C01843=1138.601,45.378,-51.505,-179.902,6.447,149.146
C01844=1138.595,45.628,-51.520,-179.900,6.448,149.145
C01845=1138.590,45.878,-51.536,-179.897,6.449,149.145
C01846=1138.585,46.127,-51.551,-179.895,6.450,149.144
C01847=1138.580,46.377,-51.567,-179.892,6.451,149.144
C01848=1138.576,46.626,-51.582,-179.890,6.452,149.143
C01849=1138.570,46.875,-51.597,-179.886,6.453,149.143
C01850=1138.565,47.125,-51.613,-179.884,6.454,149.142
C01851=1138.560,47.374,-51.628,-179.881,6.456,149.142
C01852=1138.556,47.624,-51.644,-179.879,6.456,149.141
C01853=1138.550,47.873,-51.659,-179.876,6.458,149.141
C01854=1138.546,48.122,-51.674,-179.873,6.460,149.140
C01855=1138.540,48.372,-51.690,-179.871,6.460,149.140
C01856=1138.535,48.621,-51.706,-179.868,6.462,149.139
C01857=1138.531,48.871,-51.721,-179.866,6.463,149.139
C01858=1138.525,49.120,-51.736,-179.863,6.464,149.138
C01859=1138.520,49.370,-51.752,-179.860,6.465,149.138
C01860=1138.515,49.619,-51.767,-179.858,6.466,149.137
C01861=1138.510,49.869,-51.783,-179.855,6.467,149.137
C01862=1138.505,50.118,-51.799,-179.852,6.468,149.136
C01863=1138.500,50.368,-51.814,-179.850,6.469,149.136
C01864=1138.495,50.617,-51.829,-179.847,6.471,149.135
C01865=1138.490,50.867,-51.845,-179.844,6.472,149.135
C01866=1138.485,51.116,-51.861,-179.842,6.473,149.134
C01867=1138.480,51.365,-51.876,-179.839,6.474,149.133
C01868=1138.475,51.616,-51.892,-179.837,6.475,149.133
C01869=1138.470,51.865,-51.907,-179.834,6.477,149.133
C01870=1138.465,52.114,-51.923,-179.831,6.477,149.132
C01871=1138.459,52.364,-51.938,-179.828,6.479,149.131
C01872=1138.456,52.613,-51.954,-179.826,6.480,149.131
C01873=1138.450,52.862,-51.970,-179.823,6.481,149.131
C01874=1138.445,53.131,-51.987,-179.820,6.483,149.130
C01875=1138.439,53.399,-52.004,-179.817,6.484,149.129
C01876=1138.433,53.668,-52.020,-179.815,6.485,149.129
C01877=1138.428,53.938,-52.038,-179.812,6.486,149.128
C01878=1138.423,54.186,-52.054,-179.809,6.488,149.128
C01879=1138.418,54.435,-52.069,-179.807,6.488,149.127
C01880=1138.414,54.686,-52.085,-179.804,6.490,149.127
C01881=1138.408,54.935,-52.101,-179.801,6.491,149.126
C01882=1138.403,55.184,-52.116,-179.799,6.492,149.126
C01883=1138.398,55.434,-52.133,-179.796,6.494,149.125
C01884=1138.393,55.683,-52.148,-179.793,6.494,149.125
C01885=1138.388,55.933,-52.164,-179.790,6.496,149.124
C01886=1138.384,56.182,-52.179,-179.788,6.497,149.124
C01887=1138.379,56.431,-52.196,-179.785,6.498,149.123
C01888=1138.373,56.681,-52.211,-179.782,6.500,149.123
C01889=1138.368,56.931,-52.227,-179.780,6.501,149.122
C01890=1138.363,57.180,-52.244,-179.777,6.502,149.122
C01891=1138.359,57.430,-52.260,-179.775,6.503,149.121
C01892=1138.353,57.679,-52.275,-179.772,6.504,149.121
C01893=1138.348,57.928,-52.291,-179.769,6.506,149.120
C01894=1138.343,58.178,-52.307,-179.767,6.506,149.119
C01895=1138.338,58.427,-52.323,-179.764,6.508,149.119
C01896=1138.333,58.676,-52.339,-179.762,6.509,149.119
C01897=1138.328,58.926,-52.355,-179.759,6.511,149.118
C01898=1138.323,59.175,-52.372,-179.756,6.512,149.117
C01899=1138.318,59.425,-52.387,-179.753,6.513,149.117
C01900=1138.313,59.675,-52.403,-179.751,6.514,149.117
C01901=1138.308,59.924,-52.420,-179.747,6.516,149.116
C01902=1138.303,60.173,-52.435,-179.745,6.516,149.116
C01903=1138.298,60.422,-52.452,-179.743,6.518,149.115
C01904=1138.293,60.672,-52.468,-179.740,6.519,149.115
C01905=1138.288,60.921,-52.484,-179.737,6.520,149.114
C01906=1138.283,61.171,-52.500,-179.734,6.522,149.114
C01907=1138.278,61.420,-52.516,-179.732,6.523,149.113
C01908=1138.273,61.670,-52.532,-179.729,6.524,149.112
C01909=1138.268,61.919,-52.548,-179.726,6.526,149.112
C01910=1138.263,62.169,-52.564,-179.724,6.526,149.112
C01911=1138.258,62.418,-52.581,-179.721,6.528,149.111
C01912=1138.254,62.668,-52.597,-179.719,6.529,149.110
C01913=1138.248,62.917,-52.613,-179.716,6.530,149.110
C01914=1138.244,63.167,-52.629,-179.713,6.532,149.110
C01915=1138.239,63.416,-52.645,-179.711,6.532,149.109
C01916=1138.234,63.666,-52.661,-179.708,6.534,149.108
C01917=1138.229,63.914,-52.677,-179.705,6.536,149.108
C01918=1138.224,64.164,-52.694,-179.703,6.536,149.108
C01919=1138.219,64.413,-52.710,-179.700,6.538,149.107
C01920=1138.214,64.663,-52.727,-179.697,6.539,149.106
C01921=1138.208,64.912,-52.743,-179.695,6.540,149.106
C01922=1138.204,65.162,-52.759,-179.692,6.542,149.105
C01923=1138.199,65.411,-52.776,-179.689,6.543,149.105
C01924=1138.194,65.661,-52.791,-179.687,6.544,149.105
C01925=1138.189,65.910,-52.808,-179.684,6.546,149.104
C01926=1138.184,66.159,-52.824,-179.681,6.547,149.103
C01927=1138.178,66.409,-52.841,-179.679,6.548,149.103
C01928=1138.174,66.658,-52.857,-179.676,6.549,149.103
C01929=1138.169,66.908,-52.874,-179.673,6.551,149.102
C01930=1138.164,67.157,-52.890,-179.670,6.552,149.101
C01931=1138.159,67.407,-52.906,-179.668,6.553,149.101
C01932=1138.154,67.655,-52.923,-179.665,6.555,149.101
C01933=1138.149,67.905,-52.940,-179.662,6.555,149.100
C01934=1138.144,68.154,-52.956,-179.659,6.557,149.099
C01935=1138.139,68.404,-52.972,-179.657,6.559,149.099
C01936=1138.135,68.654,-52.989,-179.655,6.559,149.099
C01937=1138.129,68.903,-53.006,-179.651,6.561,149.098
C01938=1138.124,69.152,-53.022,-179.649,6.562,149.098
C01939=1138.119,69.402,-53.038,-179.646,6.564,149.097
C01940=1138.115,69.651,-53.055,-179.644,6.565,149.097
C01941=1138.109,69.901,-53.072,-179.640,6.566,149.096
C01942=1138.104,70.150,-53.088,-179.638,6.568,149.096
C01943=1138.100,70.399,-53.105,-179.636,6.569,149.095
C01944=1138.095,70.648,-53.121,-179.633,6.570,149.095
C01945=1138.089,70.898,-53.138,-179.630,6.572,149.094
C01946=1138.085,71.148,-53.154,-179.627,6.572,149.094
C01947=1138.080,71.397,-53.171,-179.625,6.574,149.093
C01948=1138.074,71.646,-53.188,-179.622,6.576,149.093
C01949=1138.070,71.896,-53.205,-179.619,6.577,149.092
C01950=1138.065,72.145,-53.221,-179.617,6.578,149.092
C01951=1138.060,72.394,-53.238,-179.614,6.580,149.091
C01952=1138.055,72.644,-53.255,-179.611,6.581,149.091
C01953=1138.050,72.893,-53.271,-179.608,6.582,149.090
C01954=1138.045,73.143,-53.288,-179.606,6.583,149.090
C01955=1138.040,73.392,-53.305,-179.603,6.585,149.089
C01956=1138.035,73.641,-53.321,-179.600,6.587,149.089
C01957=1138.030,73.891,-53.339,-179.598,6.587,149.088
C01958=1138.026,74.140,-53.355,-179.595,6.589,149.088
C01959=1138.020,74.389,-53.372,-179.592,6.590,149.087
C01960=1138.015,74.639,-53.389,-179.590,6.591,149.087
C01961=1138.011,74.888,-53.405,-179.587,6.593,149.086
C01962=1138.006,75.138,-53.423,-179.584,6.594,149.086
C01963=1138.001,75.387,-53.439,-179.581,6.596,149.085
C01964=1137.995,75.637,-53.456,-179.579,6.597,149.085
C01965=1137.991,75.886,-53.473,-179.576,6.598,149.084
C01966=1137.985,76.135,-53.490,-179.573,6.600,149.084
C01967=1137.981,76.385,-53.507,-179.570,6.601,149.083
C01968=1137.976,76.634,-53.523,-179.568,6.602,149.083
C01969=1137.971,76.884,-53.540,-179.565,6.604,149.082
C01970=1137.966,77.132,-53.557,-179.562,6.605,149.082
C01971=1137.961,77.382,-53.575,-179.559,6.607,149.081
C01972=1137.956,77.631,-53.591,-179.557,6.608,149.081
C01973=1137.951,77.881,-53.609,-179.555,6.609,149.081
C01974=1137.946,78.130,-53.625,-179.551,6.611,149.080
C01975=1137.941,78.380,-53.642,-179.549,6.612,149.080
C01976=1137.937,78.629,-53.660,-179.546,6.613,149.079
C01977=1137.931,78.878,-53.677,-179.544,6.615,149.079
C01978=1137.926,79.146,-53.695,-179.540,6.616,149.078
C01979=1137.921,79.415,-53.713,-179.538,6.618,149.078
C01980=1137.915,79.684,-53.732,-179.535,6.619,149.077
C01981=1137.910,79.952,-53.750,-179.532,6.621,149.077
C01982=1137.905,80.202,-53.767,-179.529,6.622,149.076
C01983=1137.901,80.450,-53.784,-179.526,6.624,149.076
C01984=1137.896,80.700,-53.802,-179.524,6.624,149.075
C01985=1137.890,80.949,-53.819,-179.521,6.626,149.075
C01986=1137.885,81.199,-53.835,-179.518,6.628,149.074
C01987=1137.880,81.448,-53.853,-179.515,6.629,149.074
C01988=1137.876,81.698,-53.870,-179.513,6.631,149.073
C01989=1137.871,81.947,-53.887,-179.510,6.632,149.073
C01990=1137.866,82.196,-53.905,-179.507,6.633,149.072
C01991=1137.861,82.445,-53.921,-179.505,6.635,149.072
C01992=1137.855,82.695,-53.939,-179.502,6.637,149.071
C01993=1137.851,82.944,-53.957,-179.499,6.637,149.071
C01994=1137.846,83.194,-53.973,-179.496,6.639,149.070
C01995=1137.841,83.443,-53.991,-179.494,6.640,149.070
C01996=1137.837,83.692,-54.008,-179.491,6.642,149.069
C01997=1137.831,83.942,-54.025,-179.488,6.644,149.069
C01998=1137.826,84.191,-54.043,-179.486,6.644,149.068
C01999=1137.821,84.440,-54.060,-179.483,6.646,149.068
C02000=1137.817,84.689,-54.078,-179.480,6.648,149.068
C02001=1137.811,84.939,-54.095,-179.477,6.649,149.067
C02002=1137.806,85.188,-54.113,-179.475,6.651,149.067
C02003=1137.802,85.438,-54.129,-179.472,6.651,149.066
C02004=1137.797,85.687,-54.147,-179.469,6.653,149.066
C02005=1137.792,85.937,-54.165,-179.466,6.655,149.065
C02006=1137.788,86.186,-54.182,-179.464,6.656,149.065
C02007=1137.782,86.435,-54.199,-179.461,6.658,149.064
C02008=1137.778,86.685,-54.217,-179.458,6.659,149.064
C02009=1137.772,86.934,-54.234,-179.456,6.660,149.063
C02010=1137.768,87.183,-54.252,-179.453,6.662,149.063
C02011=1137.762,87.432,-54.269,-179.450,6.663,149.062
C02012=1137.757,87.681,-54.287,-179.447,6.665,149.062
C02013=1137.752,87.931,-54.304,-179.444,6.666,149.061
C02014=1137.747,88.180,-54.322,-179.441,6.668,149.061
C02015=1137.743,88.429,-54.339,-179.439,6.669,149.060
C02016=1137.738,88.679,-54.357,-179.437,6.671,149.060
C02017=1137.733,88.928,-54.375,-179.434,6.672,149.060
C02018=1137.728,89.178,-54.392,-179.431,6.674,149.059
C02019=1137.723,89.427,-54.410,-179.428,6.675,149.059
C02020=1137.719,89.676,-54.427,-179.425,6.677,149.058
C02021=1137.713,89.926,-54.445,-179.423,6.678,149.058
C02022=1137.709,90.175,-54.463,-179.420,6.679,149.057
C02023=1137.704,90.424,-54.481,-179.417,6.681,149.057
C02024=1137.698,90.674,-54.498,-179.414,6.682,149.056
C02025=1137.693,90.923,-54.516,-179.412,6.684,149.056
C02026=1137.689,91.172,-54.534,-179.409,6.686,149.055
C02027=1137.684,91.421,-54.551,-179.406,6.687,149.055
C02028=1137.679,91.671,-54.568,-179.404,6.688,149.055
C02029=1137.674,91.920,-54.586,-179.401,6.690,149.054
C02030=1137.669,92.169,-54.604,-179.398,6.691,149.053
C02031=1137.664,92.419,-54.622,-179.395,6.693,149.053
C02032=1137.659,92.668,-54.640,-179.392,6.695,149.053
C02033=1137.654,92.918,-54.658,-179.390,6.696,149.052
C02034=1137.649,93.167,-54.676,-179.387,6.698,149.052
C02035=1137.644,93.416,-54.694,-179.385,6.699,149.051
C02036=1137.640,93.665,-54.712,-179.382,6.700,149.051
C02037=1137.635,93.916,-54.729,-179.379,6.702,149.050
C02038=1137.630,94.165,-54.747,-179.376,6.703,149.050
C02039=1137.625,94.414,-54.765,-179.373,6.705,149.049
C02040=1137.620,94.663,-54.783,-179.371,6.707,149.049
C02041=1137.615,94.912,-54.801,-179.368,6.708,149.049
C02042=1137.610,95.161,-54.819,-179.365,6.710,149.048
C02043=1137.605,95.411,-54.837,-179.362,6.711,149.048
C02044=1137.600,95.660,-54.854,-179.360,6.712,149.047
C02045=1137.595,95.910,-54.872,-179.357,6.714,149.047
C02046=1137.590,96.159,-54.890,-179.354,6.716,149.046
C02047=1137.586,96.408,-54.908,-179.352,6.717,149.046
C02048=1137.581,96.658,-54.927,-179.349,6.719,149.045
C02049=1137.576,96.907,-54.945,-179.346,6.720,149.045
C02050=1137.571,97.156,-54.963,-179.343,6.722,149.044
C02051=1137.566,97.405,-54.981,-179.340,6.724,149.044
C02052=1137.562,97.655,-54.999,-179.337,6.725,149.044
C02053=1137.557,97.904,-55.017,-179.335,6.726,149.043
C02054=1137.552,98.153,-55.035,-179.333,6.728,149.043
C02055=1137.547,98.403,-55.053,-179.330,6.729,149.042
C02056=1137.543,98.652,-55.071,-179.327,6.731,149.042
C02057=1137.538,98.901,-55.089,-179.324,6.732,149.041
C02058=1137.532,99.151,-55.107,-179.321,6.734,149.041
C02059=1137.527,99.400,-55.125,-179.318,6.736,149.040
C02060=1137.522,99.649,-55.143,-179.316,6.737,149.040
C02061=1137.518,99.898,-55.162,-179.313,6.739,149.040
C02062=1137.513,100.147,-55.180,-179.310,6.741,149.039
C02063=1137.508,100.397,-55.198,-179.307,6.742,149.039
C02064=1137.503,100.646,-55.216,-179.304,6.744,149.038
C02065=1137.498,100.895,-55.235,-179.301,6.745,149.038
C02066=1137.493,101.145,-55.253,-179.299,6.746,149.037
C02067=1137.489,101.394,-55.271,-179.297,6.748,149.037
C02068=1137.484,101.643,-55.289,-179.294,6.750,149.036
C02069=1137.479,101.892,-55.308,-179.291,6.751,149.036
C02070=1137.474,102.141,-55.326,-179.288,6.753,149.036
C02071=1137.469,102.391,-55.345,-179.286,6.755,149.035
C02072=1137.464,102.641,-55.363,-179.282,6.756,149.035
C02073=1137.459,102.890,-55.381,-179.280,6.758,149.034
C02074=1137.455,103.138,-55.399,-179.277,6.759,149.034
C02075=1137.450,103.389,-55.418,-179.274,6.761,149.033
C02076=1137.445,103.638,-55.436,-179.272,6.763,149.033
C02077=1137.440,103.887,-55.454,-179.269,6.764,149.033
C02078=1137.435,104.135,-55.473,-179.266,6.766,149.032
C02079=1137.430,104.386,-55.492,-179.263,6.768,149.032
C02080=1137.425,104.635,-55.510,-179.261,6.769,149.031
C02081=1137.421,104.883,-55.529,-179.257,6.771,149.031
C02082=1137.415,105.152,-55.549,-179.255,6.772,149.030
C02083=1137.410,105.421,-55.568,-179.252,6.774,149.030
C02084=1137.404,105.689,-55.588,-179.249,6.776,149.029
C02085=1137.400,105.957,-55.609,-179.246,6.777,149.029
C02086=1137.395,106.206,-55.627,-179.243,6.779,149.028
C02087=1137.390,106.456,-55.646,-179.240,6.780,149.028
C02088=1137.385,106.705,-55.664,-179.238,6.782,149.028
C02089=1137.380,106.954,-55.682,-179.235,6.784,149.027
C02090=1137.375,107.204,-55.702,-179.232,6.785,149.027
C02091=1137.371,107.453,-55.720,-179.230,6.787,149.026
C02092=1137.366,107.702,-55.738,-179.227,6.789,149.026
C02093=1137.361,107.952,-55.757,-179.224,6.790,149.025
C02094=1137.356,108.201,-55.775,-179.221,6.792,149.025
C02095=1137.351,108.450,-55.795,-179.218,6.793,149.024
C02096=1137.346,108.700,-55.813,-179.215,6.795,149.024
C02097=1137.342,108.948,-55.832,-179.213,6.797,149.024
C02098=1137.336,109.198,-55.850,-179.210,6.798,149.023
C02099=1137.332,109.447,-55.869,-179.207,6.800,149.023
C02100=1137.326,109.696,-55.888,-179.204,6.802,149.022
C02101=1137.322,109.946,-55.907,-179.202,6.804,149.022
C02102=1137.317,110.195,-55.926,-179.199,6.805,149.022
C02103=1137.312,110.444,-55.944,-179.196,6.807,149.021
C02104=1137.308,110.694,-55.963,-179.194,6.809,149.021
C02105=1137.302,110.942,-55.982,-179.191,6.810,149.020
C02106=1137.298,111.192,-56.001,-179.188,6.812,149.020
C02107=1137.293,111.441,-56.020,-179.185,6.813,149.019
C02108=1137.288,111.690,-56.038,-179.182,6.815,149.019
C02109=1137.283,111.940,-56.057,-179.179,6.817,149.019
C02110=1137.279,112.188,-56.076,-179.177,6.818,149.018
C02111=1137.274,112.438,-56.096,-179.174,6.820,149.018
C02112=1137.269,112.687,-56.114,-179.171,6.822,149.017
C02113=1137.264,112.936,-56.133,-179.168,6.823,149.017
C02114=1137.259,113.186,-56.153,-179.166,6.825,149.016
C02115=1137.254,113.435,-56.171,-179.163,6.827,149.016
C02116=1137.249,113.684,-56.190,-179.160,6.828,149.016
C02117=1137.245,113.933,-56.209,-179.158,6.830,149.015
C02118=1137.240,114.183,-56.228,-179.154,6.833,149.015
C02119=1137.235,114.432,-56.246,-179.152,6.834,149.014
C02120=1137.230,114.681,-56.266,-179.149,6.836,149.014
C02121=1137.225,114.930,-56.285,-179.146,6.838,149.014
C02122=1137.221,115.180,-56.304,-179.143,6.839,149.013
C02123=1137.215,115.429,-56.323,-179.141,6.841,149.013
C02124=1137.211,115.678,-56.342,-179.137,6.842,149.012
C02125=1137.206,115.927,-56.361,-179.135,6.844,149.012
C02126=1137.201,116.177,-56.381,-179.132,6.846,149.011
C02127=1137.196,116.426,-56.399,-179.129,6.847,149.011
C02128=1137.191,116.675,-56.419,-179.126,6.849,149.011
C02129=1137.186,116.924,-56.438,-179.124,6.851,149.010
C02130=1137.182,117.173,-56.457,-179.121,6.852,149.010
C02131=1137.177,117.422,-56.476,-179.118,6.854,149.009
C02132=1137.172,117.672,-56.496,-179.116,6.856,149.009
C02133=1137.167,117.920,-56.515,-179.113,6.857,149.009
C02134=1137.163,118.170,-56.534,-179.110,6.859,149.008
C02135=1137.157,118.419,-56.553,-179.107,6.861,149.008
C02136=1137.153,118.669,-56.572,-179.105,6.862,149.007
C02137=1137.148,118.918,-56.591,-179.101,6.865,149.007
C02138=1137.143,119.167,-56.611,-179.099,6.867,149.007
C02139=1137.139,119.416,-56.630,-179.096,6.868,149.006
C02140=1137.134,119.665,-56.649,-179.093,6.870,149.006
C02141=1137.129,119.915,-56.669,-179.090,6.872,149.005
C02142=1137.123,120.164,-56.688,-179.088,6.873,149.005
C02143=1137.119,120.413,-56.707,-179.085,6.875,149.005
C02144=1137.114,120.662,-56.727,-179.082,6.877,149.004
C02145=1137.109,120.911,-56.746,-179.079,6.878,149.004
C02146=1137.105,121.161,-56.766,-179.077,6.880,149.003
C02147=1137.099,121.410,-56.785,-179.074,6.882,149.003
C02148=1137.095,121.659,-56.804,-179.071,6.883,149.002
C02149=1137.090,121.908,-56.824,-179.068,6.886,149.002
C02150=1137.085,122.158,-56.843,-179.065,6.888,149.002
C02151=1137.081,122.406,-56.864,-179.063,6.889,149.001
C02152=1137.075,122.655,-56.883,-179.060,6.891,149.001
C02153=1137.071,122.905,-56.902,-179.057,6.893,149.000
C02154=1137.067,123.154,-56.922,-179.054,6.894,149.000
C02155=1137.061,123.403,-56.941,-179.052,6.896,149.000
C02156=1137.057,123.653,-56.961,-179.049,6.898,148.999
C02157=1137.052,123.902,-56.980,-179.046,6.899,148.999
C02158=1137.046,124.151,-56.999,-179.043,6.901,148.998
C02159=1137.042,124.400,-57.020,-179.040,6.904,148.998
C02160=1137.038,124.649,-57.039,-179.037,6.905,148.998
C02161=1137.033,124.898,-57.058,-179.035,6.907,148.997
C02162=1137.028,125.148,-57.078,-179.032,6.909,148.997
C02163=1137.024,125.397,-57.098,-179.029,6.910,148.996
C02164=1137.018,125.645,-57.118,-179.027,6.912,148.996
C02165=1137.013,125.895,-57.137,-179.024,6.914,148.996
C02166=1137.009,126.145,-57.157,-179.021,6.915,148.995
C02167=1137.004,126.394,-57.177,-179.018,6.918,148.995
C02168=1136.999,126.642,-57.197,-179.015,6.920,148.995
C02169=1136.994,126.892,-57.216,-179.012,6.921,148.994
C02170=1136.989,127.142,-57.236,-179.010,6.923,148.994
C02171=1136.984,127.390,-57.256,-179.007,6.925,148.993
C02172=1136.980,127.639,-57.275,-179.004,6.926,148.993
C02173=1136.975,127.889,-57.295,-179.001,6.928,148.993
C02174=1136.970,128.138,-57.316,-178.998,6.931,148.992
C02175=1136.965,128.387,-57.335,-178.995,6.932,148.992
C02176=1136.961,128.636,-57.355,-178.993,6.934,148.991
C02177=1136.956,128.885,-57.375,-178.990,6.936,148.991
C02178=1136.951,129.135,-57.394,-178.987,6.937,148.991
C02179=1136.946,129.383,-57.414,-178.984,6.939,148.990
C02180=1136.941,129.633,-57.434,-178.982,6.941,148.990
C02181=1136.937,129.882,-57.455,-178.978,6.943,148.989
C02182=1136.932,130.131,-57.474,-178.976,6.945,148.989
C02183=1136.927,130.380,-57.493,-178.973,6.947,148.989
C02184=1136.922,130.629,-57.514,-178.970,6.948,148.988
C02185=1136.918,130.879,-57.533,-178.968,6.950,148.988
C02186=1136.912,131.147,-57.556,-178.964,6.953,148.987
C02187=1136.907,131.416,-57.577,-178.961,6.954,148.987
C02188=1136.903,131.684,-57.598,-178.959,6.956,148.987
C02189=1136.897,131.953,-57.620,-178.955,6.958,148.986
C02190=1136.892,132.202,-57.640,-178.953,6.960,148.986
C02191=1136.888,132.451,-57.660,-178.950,6.962,148.985
C02192=1136.883,132.700,-57.680,-178.947,6.964,148.985
C02193=1136.878,132.949,-57.700,-178.944,6.966,148.985
C02194=1136.873,133.198,-57.721,-178.941,6.968,148.984
C02195=1136.868,133.448,-57.741,-178.939,6.969,148.984
C02196=1136.864,133.697,-57.761,-178.936,6.971,148.983
C02197=1136.859,133.946,-57.781,-178.934,6.973,148.983
C02198=1136.855,134.195,-57.801,-178.930,6.976,148.983
C02199=1136.850,134.443,-57.821,-178.928,6.977,148.983
C02200=1136.844,134.693,-57.841,-178.925,6.979,148.982
C02201=1136.840,134.942,-57.862,-178.922,6.981,148.982
C02202=1136.835,135.191,-57.882,-178.919,6.982,148.981
C02203=1136.831,135.441,-57.902,-178.916,6.985,148.981
C02204=1136.825,135.690,-57.923,-178.913,6.987,148.981
C02205=1136.821,135.939,-57.943,-178.911,6.988,148.980
C02206=1136.816,136.189,-57.963,-178.908,6.990,148.980
C02207=1136.812,136.438,-57.983,-178.905,6.992,148.979
C02208=1136.806,136.686,-58.004,-178.902,6.994,148.979
C02209=1136.802,136.935,-58.024,-178.899,6.996,148.979
C02210=1136.797,137.185,-58.044,-178.897,6.998,148.978
C02211=1136.792,137.434,-58.064,-178.894,7.000,148.978
C02212=1136.787,137.683,-58.085,-178.891,7.001,148.978
C02213=1136.783,137.932,-58.106,-178.888,7.004,148.977
C02214=1136.778,138.181,-58.126,-178.885,7.006,148.977
C02215=1136.773,138.431,-58.146,-178.883,7.007,148.976
C02216=1136.768,138.680,-58.167,-178.880,7.009,148.976
C02217=1136.764,138.928,-58.187,-178.877,7.011,148.976
C02218=1136.759,139.178,-58.208,-178.874,7.013,148.975
C02219=1136.754,139.427,-58.228,-178.871,7.015,148.975
C02220=1136.750,139.676,-58.249,-178.869,7.017,148.975
C02221=1136.745,139.925,-58.270,-178.866,7.019,148.974
C02222=1136.740,140.174,-58.290,-178.863,7.021,148.974
C02223=1136.736,140.423,-58.310,-178.860,7.023,148.974
C02224=1136.730,140.673,-58.331,-178.857,7.025,148.973
C02225=1136.726,140.922,-58.351,-178.855,7.026,148.973
C02226=1136.721,141.171,-58.372,-178.851,7.029,148.972
C02227=1136.716,141.420,-58.392,-178.849,7.030,148.972
C02228=1136.712,141.669,-58.413,-178.846,7.032,148.972
C02229=1136.707,141.918,-58.434,-178.844,7.034,148.971
C02230=1136.702,142.167,-58.454,-178.840,7.037,148.971
C02231=1136.697,142.416,-58.475,-178.838,7.038,148.971
C02232=1136.693,142.665,-58.495,-178.835,7.040,148.970
C02233=1136.687,142.914,-58.516,-178.832,7.043,148.970
C02234=1136.683,143.163,-58.537,-178.829,7.044,148.970
C02235=1136.678,143.412,-58.558,-178.826,7.046,148.969
C02236=1136.674,143.661,-58.579,-178.824,7.048,148.969
C02237=1136.669,143.910,-58.599,-178.821,7.051,148.969
C02238=1136.664,144.159,-58.620,-178.818,7.052,148.968
C02239=1136.660,144.408,-58.640,-178.815,7.054,148.968
C02240=1136.655,144.658,-58.662,-178.813,7.056,148.967
C02241=1136.650,144.907,-58.683,-178.809,7.058,148.967
C02242=1136.646,145.156,-58.703,-178.807,7.060,148.967
C02243=1136.640,145.406,-58.724,-178.804,7.062,148.967
C02244=1136.636,145.654,-58.745,-178.801,7.064,148.966
C02245=1136.631,145.903,-58.766,-178.798,7.066,148.966
C02246=1136.627,146.152,-58.787,-178.796,7.068,148.965
C02247=1136.621,146.401,-58.807,-178.793,7.070,148.965
C02248=1136.617,146.650,-58.828,-178.790,7.072,148.965
C02249=1136.612,146.899,-58.850,-178.787,7.074,148.964
C02250=1136.608,147.149,-58.871,-178.785,7.076,148.964
C02251=1136.603,147.398,-58.891,-178.781,7.078,148.964
C02252=1136.598,147.647,-58.912,-178.779,7.080,148.963
C02253=1136.594,147.895,-58.933,-178.776,7.082,148.963
C02254=1136.589,148.145,-58.954,-178.773,7.083,148.963
C02255=1136.583,148.394,-58.975,-178.770,7.086,148.962
C02256=1136.580,148.643,-58.997,-178.768,7.088,148.962
C02257=1136.575,148.892,-59.018,-178.765,7.090,148.962
C02258=1136.570,149.142,-59.039,-178.762,7.092,148.961
C02259=1136.565,149.390,-59.060,-178.759,7.094,148.961
C02260=1136.560,149.639,-59.081,-178.756,7.096,148.961
C02261=1136.555,149.888,-59.102,-178.753,7.099,148.960
C02262=1136.552,150.137,-59.123,-178.751,7.100,148.960
C02263=1136.546,150.387,-59.144,-178.748,7.102,148.960
C02264=1136.542,150.635,-59.166,-178.745,7.104,148.959
C02265=1136.536,150.885,-59.187,-178.742,7.106,148.959
C02266=1136.532,151.133,-59.207,-178.739,7.108,148.958
C02267=1136.528,151.383,-59.229,-178.736,7.111,148.958
C02268=1136.522,151.632,-59.250,-178.734,7.112,148.958
C02269=1136.518,151.881,-59.272,-178.731,7.114,148.958
C02270=1136.513,152.130,-59.292,-178.728,7.117,148.957
C02271=1136.508,152.378,-59.314,-178.725,7.118,148.957
C02272=1136.504,152.628,-59.335,-178.723,7.120,148.957
C02273=1136.499,152.877,-59.357,-178.719,7.123,148.956
C02274=1136.494,153.126,-59.378,-178.717,7.125,148.956
C02275=1136.490,153.375,-59.399,-178.714,7.126,148.955
C02276=1136.485,153.624,-59.420,-178.711,7.129,148.955
C02277=1136.480,153.873,-59.442,-178.708,7.131,148.955
C02278=1136.475,154.122,-59.463,-178.706,7.133,148.955
C02279=1136.471,154.372,-59.485,-178.702,7.135,148.954
C02280=1136.467,154.620,-59.506,-178.700,7.137,148.954
C02281=1136.461,154.869,-59.527,-178.697,7.139,148.954
C02282=1136.456,155.118,-59.549,-178.694,7.141,148.953
C02283=1136.452,155.367,-59.571,-178.691,7.143,148.953
C02284=1136.447,155.617,-59.592,-178.688,7.146,148.953
C02285=1136.442,155.865,-59.613,-178.685,7.147,148.952
C02286=1136.438,156.115,-59.635,-178.683,7.149,148.952
C02287=1136.433,156.364,-59.656,-178.680,7.152,148.952
C02288=1136.429,156.612,-59.677,-178.677,7.154,148.951
C02289=1136.424,156.861,-59.700,-178.674,7.155,148.951
C02290=1136.419,157.131,-59.723,-178.671,7.158,148.951
C02291=1136.414,157.400,-59.746,-178.668,7.161,148.950
C02292=1136.408,157.668,-59.769,-178.666,7.163,148.950
C02293=1136.403,157.937,-59.793,-178.662,7.165,148.950
C02294=1136.399,158.186,-59.814,-178.660,7.167,148.949
C02295=1136.394,158.436,-59.835,-178.656,7.169,148.949
C02296=1136.390,158.685,-59.857,-178.654,7.171,148.949
C02297=1136.385,158.934,-59.879,-178.651,7.173,148.948
C02298=1136.380,159.182,-59.901,-178.648,7.176,148.948
C02299=1136.376,159.432,-59.923,-178.645,7.177,148.948
C02300=1136.371,159.680,-59.944,-178.642,7.180,148.947
C02301=1136.366,159.929,-59.965,-178.640,7.182,148.947
C02302=1136.362,160.179,-59.987,-178.637,7.184,148.947
C02303=1136.357,160.427,-60.009,-178.634,7.186,148.946
C02304=1136.352,160.677,-60.031,-178.631,7.188,148.946
C02305=1136.348,160.925,-60.053,-178.628,7.191,148.946
C02306=1136.343,161.175,-60.075,-178.625,7.192,148.945
C02307=1136.338,161.424,-60.097,-178.622,7.195,148.945
C02308=1136.333,161.672,-60.119,-178.620,7.197,148.945
C02309=1136.329,161.922,-60.141,-178.617,7.199,148.945
C02310=1136.324,162.170,-60.162,-178.614,7.201,148.944
C02311=1136.319,162.420,-60.184,-178.612,7.203,148.944
C02312=1136.315,162.668,-60.206,-178.608,7.206,148.944
C02313=1136.310,162.918,-60.228,-178.606,7.207,148.943
C02314=1136.305,163.166,-60.250,-178.603,7.209,148.943
C02315=1136.301,163.416,-60.272,-178.600,7.212,148.943
C02316=1136.296,163.664,-60.294,-178.597,7.214,148.942
C02317=1136.291,163.914,-60.316,-178.594,7.216,148.942
C02318=1136.286,164.163,-60.338,-178.592,7.218,148.942
C02319=1136.282,164.412,-60.360,-178.589,7.221,148.942
C02320=1136.277,164.661,-60.382,-178.586,7.223,148.941
C02321=1136.273,164.910,-60.404,-178.583,7.224,148.941
C02322=1136.268,165.159,-60.425,-178.580,7.227,148.941
C02323=1136.263,165.408,-60.448,-178.578,7.229,148.940
C02324=1136.259,165.656,-60.470,-178.574,7.231,148.940
C02325=1136.254,165.906,-60.492,-178.572,7.234,148.940
C02326=1136.249,166.154,-60.514,-178.569,7.236,148.939
C02327=1136.245,166.403,-60.536,-178.566,7.238,148.939
C02328=1136.240,166.652,-60.558,-178.563,7.241,148.939
C02329=1136.235,166.902,-60.581,-178.561,7.242,148.939
C02330=1136.231,167.150,-60.603,-178.557,7.245,148.938
C02331=1136.226,167.399,-60.625,-178.555,7.247,148.938
C02332=1136.221,167.648,-60.647,-178.552,7.249,148.938
C02333=1136.217,167.897,-60.669,-178.549,7.251,148.937
C02334=1136.213,168.146,-60.692,-178.547,7.253,148.937
C02335=1136.207,168.395,-60.714,-178.543,7.256,148.937
C02336=1136.203,168.644,-60.736,-178.541,7.258,148.936
C02337=1136.198,168.893,-60.758,-178.538,7.260,148.936
C02338=1136.194,169.142,-60.781,-178.535,7.262,148.936
C02339=1136.188,169.391,-60.803,-178.532,7.265,148.936
C02340=1136.184,169.640,-60.825,-178.530,7.267,148.935
C02341=1136.179,169.889,-60.849,-178.526,7.269,148.935
C02342=1136.174,170.138,-60.870,-178.524,7.271,148.935
C02343=1136.170,170.387,-60.892,-178.521,7.274,148.935
C02344=1136.165,170.635,-60.915,-178.518,7.276,148.934
C02345=1136.161,170.885,-60.937,-178.515,7.278,148.934
C02346=1136.157,171.134,-60.960,-178.513,7.280,148.934
C02347=1136.151,171.382,-60.982,-178.509,7.283,148.933
C02348=1136.147,171.632,-61.004,-178.507,7.284,148.933
C02349=1136.142,171.881,-61.028,-178.504,7.287,148.933
C02350=1136.137,172.129,-61.049,-178.501,7.289,148.932
C02351=1136.133,172.378,-61.072,-178.498,7.292,148.932
C02352=1136.128,172.628,-61.095,-178.496,7.294,148.932
C02353=1136.124,172.876,-61.117,-178.492,7.296,148.932
C02354=1136.119,173.126,-61.140,-178.490,7.298,148.931
C02355=1136.115,173.374,-61.163,-178.487,7.301,148.931
C02356=1136.109,173.623,-61.185,-178.484,7.302,148.931
C02357=1136.105,173.872,-61.208,-178.481,7.305,148.931
C02358=1136.100,174.122,-61.230,-178.479,7.307,148.930
C02359=1136.096,174.370,-61.253,-178.475,7.310,148.930
C02360=1136.091,174.619,-61.276,-178.473,7.312,148.930
C02361=1136.087,174.868,-61.298,-178.470,7.314,148.929
C02362=1136.082,175.117,-61.322,-178.467,7.316,148.929
C02363=1136.077,175.366,-61.343,-178.464,7.319,148.929
C02364=1136.072,175.615,-61.367,-178.461,7.320,148.929
C02365=1136.068,175.863,-61.389,-178.459,7.323,148.928
C02366=1136.063,176.112,-61.412,-178.456,7.325,148.928
C02367=1136.059,176.361,-61.434,-178.453,7.328,148.928
C02368=1136.054,176.610,-61.458,-178.450,7.330,148.928
C02369=1136.050,176.859,-61.480,-178.447,7.332,148.927
C02370=1136.045,177.108,-61.503,-178.445,7.334,148.927
C02371=1136.040,177.357,-61.526,-178.442,7.337,148.927
C02372=1136.036,177.606,-61.549,-178.439,7.340,148.927
C02373=1136.031,177.855,-61.572,-178.436,7.341,148.926
C02374=1136.027,178.104,-61.594,-178.433,7.344,148.926
C02375=1136.022,178.352,-61.617,-178.431,7.346,148.926
C02376=1136.017,178.601,-61.641,-178.427,7.349,148.925
C02377=1136.013,178.851,-61.663,-178.425,7.351,148.925
C02378=1136.008,179.100,-61.686,-178.422,7.353,148.925
C02379=1136.003,179.349,-61.709,-178.419,7.355,148.925
C02380=1135.999,179.597,-61.732,-178.416,7.358,148.924
C02381=1135.994,179.846,-61.755,-178.413,7.360,148.924
C02382=1135.989,180.095,-61.779,-178.411,7.362,148.924
C02383=1135.985,180.344,-61.801,-178.407,7.365,148.924
C02384=1135.980,180.593,-61.824,-178.405,7.367,148.923
C02385=1135.976,180.842,-61.847,-178.402,7.370,148.923
C02386=1135.971,181.090,-61.870,-178.400,7.372,148.923
C02387=1135.966,181.339,-61.893,-178.396,7.374,148.923
C02388=1135.962,181.588,-61.916,-178.394,7.376,148.922
C02389=1135.958,181.837,-61.939,-178.391,7.379,148.922
C02390=1135.953,182.086,-61.963,-178.388,7.381,148.922
C02391=1135.948,182.335,-61.986,-178.385,7.383,148.922
C02392=1135.944,182.584,-62.009,-178.382,7.386,148.921
C02393=1135.939,182.832,-62.032,-178.380,7.388,148.921
C02394=1135.934,183.103,-62.057,-178.376,7.391,148.921
C02395=1135.929,183.372,-62.082,-178.374,7.393,148.921
C02396=1135.924,183.641,-62.108,-178.370,7.396,148.920
C02397=1135.919,183.911,-62.133,-178.367,7.398,148.920
C02398=1135.915,184.160,-62.156,-178.364,7.401,148.920
C02399=1135.910,184.409,-62.179,-178.362,7.403,148.919
C02400=1135.905,184.658,-62.202,-178.359,7.406,148.919
C02401=1135.901,184.907,-62.226,-178.356,7.408,148.919
C02402=1135.896,185.156,-62.249,-178.353,7.411,148.919
C02403=1135.891,185.405,-62.272,-178.350,7.413,148.918
C02404=1135.887,185.654,-62.296,-178.348,7.415,148.918
C02405=1135.883,185.902,-62.319,-178.344,7.418,148.918
C02406=1135.878,186.151,-62.343,-178.342,7.420,148.918
C02407=1135.873,186.400,-62.366,-178.339,7.422,148.918
C02408=1135.868,186.649,-62.389,-178.336,7.425,148.917
C02409=1135.863,186.898,-62.412,-178.333,7.427,148.917
C02410=1135.859,187.146,-62.436,-178.331,7.430,148.917
C02411=1135.854,187.395,-62.460,-178.328,7.432,148.917
C02412=1135.850,187.644,-62.483,-178.325,7.434,148.916
C02413=1135.845,187.893,-62.506,-178.322,7.437,148.916
C02414=1135.841,188.142,-62.531,-178.320,7.439,148.916
C02415=1135.836,188.391,-62.554,-178.316,7.442,148.916
C02416=1135.831,188.640,-62.577,-178.313,7.445,148.916
C02417=1135.827,188.888,-62.601,-178.311,7.446,148.915
C02418=1135.822,189.137,-62.625,-178.308,7.449,148.915
C02419=1135.817,189.386,-62.648,-178.305,7.452,148.915
C02420=1135.813,189.635,-62.671,-178.302,7.454,148.915
C02421=1135.808,189.884,-62.695,-178.299,7.456,148.914
C02422=1135.804,190.133,-62.719,-178.297,7.458,148.914
C02423=1135.800,190.382,-62.743,-178.294,7.461,148.914
C02424=1135.795,190.631,-62.767,-178.291,7.464,148.914
C02425=1135.790,190.880,-62.790,-178.288,7.466,148.913
C02426=1135.786,191.128,-62.814,-178.285,7.468,148.913
C02427=1135.781,191.377,-62.837,-178.282,7.471,148.913
C02428=1135.777,191.626,-62.862,-178.280,7.473,148.913
C02429=1135.772,191.875,-62.885,-178.277,7.476,148.913
C02430=1135.768,192.123,-62.909,-178.274,7.478,148.912
C02431=1135.763,192.372,-62.932,-178.271,7.481,148.912
C02432=1135.759,192.621,-62.956,-178.268,7.483,148.912
C02433=1135.753,192.870,-62.980,-178.265,7.486,148.912
C02434=1135.749,193.118,-63.004,-178.263,7.488,148.911
C02435=1135.744,193.367,-63.028,-178.260,7.491,148.911
C02436=1135.740,193.616,-63.052,-178.256,7.493,148.911
C02437=1135.736,193.865,-63.076,-178.254,7.495,148.911
C02438=1135.731,194.114,-63.100,-178.251,7.498,148.911
C02439=1135.727,194.363,-63.123,-178.248,7.501,148.910
C02440=1135.721,194.612,-63.148,-178.246,7.503,148.910
C02441=1135.717,194.860,-63.172,-178.243,7.505,148.910
C02442=1135.712,195.109,-63.195,-178.240,7.508,148.910
C02443=1135.708,195.357,-63.219,-178.237,7.510,148.909
C02444=1135.704,195.607,-63.243,-178.234,7.513,148.909
C02445=1135.699,195.856,-63.268,-178.231,7.516,148.909
C02446=1135.694,196.104,-63.292,-178.228,7.518,148.909
C02447=1135.690,196.353,-63.316,-178.226,7.520,148.909
C02448=1135.685,196.602,-63.339,-178.223,7.523,148.908
C02449=1135.681,196.850,-63.363,-178.220,7.526,148.908
C02450=1135.676,197.100,-63.388,-178.218,7.528,148.908
C02451=1135.672,197.349,-63.412,-178.214,7.530,148.908
C02452=1135.667,197.597,-63.436,-178.212,7.533,148.908
C02453=1135.662,197.846,-63.460,-178.209,7.535,148.907
C02454=1135.658,198.094,-63.484,-178.206,7.538,148.907
C02455=1135.654,198.344,-63.508,-178.203,7.541,148.907
C02456=1135.649,198.592,-63.532,-178.200,7.543,148.907
C02457=1135.644,198.841,-63.557,-178.198,7.545,148.907
C02458=1135.640,199.090,-63.581,-178.194,7.548,148.906
C02459=1135.636,199.339,-63.605,-178.192,7.551,148.906
C02460=1135.631,199.587,-63.630,-178.189,7.553,148.906
C02461=1135.626,199.836,-63.654,-178.186,7.555,148.906
C02462=1135.622,200.085,-63.677,-178.183,7.558,148.906
C02463=1135.617,200.334,-63.702,-178.180,7.561,148.905
C02464=1135.613,200.583,-63.727,-178.178,7.563,148.905
C02465=1135.608,200.831,-63.751,-178.175,7.566,148.905
C02466=1135.603,201.080,-63.775,-178.172,7.569,148.905
C02467=1135.599,201.329,-63.800,-178.169,7.571,148.904
C02468=1135.594,201.578,-63.824,-178.167,7.573,148.904
C02469=1135.590,201.826,-63.848,-178.163,7.576,148.904
C02470=1135.585,202.075,-63.874,-178.161,7.579,148.904
C02471=1135.581,202.324,-63.898,-178.158,7.582,148.904
C02472=1135.577,202.572,-63.922,-178.155,7.583,148.903
C02473=1135.572,202.822,-63.947,-178.152,7.586,148.903
C02474=1135.568,203.070,-63.971,-178.149,7.589,148.903
C02475=1135.562,203.319,-63.995,-178.146,7.592,148.903
C02476=1135.559,203.568,-64.020,-178.144,7.594,148.903
C02477=1135.554,203.817,-64.045,-178.141,7.597,148.903
C02478=1135.549,204.065,-64.069,-178.138,7.599,148.902
C02479=1135.545,204.315,-64.094,-178.135,7.602,148.902
C02480=1135.540,204.563,-64.118,-178.133,7.604,148.902
C02481=1135.535,204.811,-64.143,-178.129,7.607,148.902
C02482=1135.532,205.060,-64.168,-178.127,7.610,148.902
C02483=1135.526,205.309,-64.192,-178.124,7.613,148.902
C02484=1135.521,205.558,-64.217,-178.121,7.614,148.901
C02485=1135.518,205.807,-64.241,-178.118,7.617,148.901
C02486=1135.512,206.055,-64.266,-178.116,7.620,148.901
C02487=1135.509,206.304,-64.291,-178.113,7.623,148.901
C02488=1135.504,206.553,-64.316,-178.109,7.626,148.901
C02489=1135.499,206.801,-64.340,-178.107,7.628,148.900
C02490=1135.495,207.050,-64.365,-178.104,7.631,148.900
C02491=1135.490,207.299,-64.390,-178.101,7.633,148.900
C02492=1135.486,207.548,-64.415,-178.098,7.636,148.900
C02493=1135.481,207.796,-64.439,-178.096,7.638,148.900
C02494=1135.476,208.045,-64.464,-178.093,7.641,148.900
C02495=1135.473,208.294,-64.489,-178.090,7.644,148.899
C02496=1135.467,208.542,-64.514,-178.087,7.646,148.899
C02497=1135.463,208.792,-64.539,-178.084,7.649,148.899
C02498=1135.458,209.062,-64.566,-178.081,7.652,148.899
C02499=1135.453,209.332,-64.593,-178.078,7.655,148.899
C02500=1135.449,209.603,-64.621,-178.075,7.658,148.899
C02501=1135.444,209.873,-64.647,-178.072,7.660,148.898
C02502=1135.439,210.123,-64.672,-178.069,7.663,148.898
C02503=1135.434,210.371,-64.697,-178.067,7.666,148.898
C02504=1135.430,210.620,-64.723,-178.063,7.669,148.898
C02505=1135.425,210.869,-64.747,-178.061,7.671,148.898
C02506=1135.421,211.117,-64.773,-178.058,7.674,148.898
C02507=1135.416,211.366,-64.797,-178.055,7.676,148.897
C02508=1135.412,211.615,-64.823,-178.052,7.679,148.897
C02509=1135.407,211.863,-64.847,-178.049,7.682,148.897
C02510=1135.403,212.112,-64.873,-178.047,7.685,148.897
C02511=1135.398,212.361,-64.897,-178.044,7.687,148.897
C02512=1135.394,212.610,-64.923,-178.041,7.689,148.896
C02513=1135.390,212.858,-64.947,-178.038,7.692,148.896
C02514=1135.385,213.107,-64.973,-178.035,7.695,148.896
C02515=1135.380,213.355,-64.998,-178.033,7.698,148.896
C02516=1135.376,213.604,-65.023,-178.030,7.700,148.896
C02517=1135.371,213.853,-65.049,-178.027,7.703,148.896
C02518=1135.367,214.102,-65.074,-178.024,7.706,148.896
C02519=1135.363,214.350,-65.099,-178.021,7.709,148.896
C02520=1135.358,214.599,-65.124,-178.019,7.711,148.895
C02521=1135.354,214.848,-65.149,-178.015,7.714,148.895
C02522=1135.349,215.096,-65.175,-178.013,7.717,148.895
C02523=1135.345,215.345,-65.201,-178.010,7.719,148.895
C02524=1135.340,215.594,-65.225,-178.008,7.722,148.895
C02525=1135.335,215.842,-65.251,-178.005,7.725,148.895
C02526=1135.331,216.091,-65.277,-178.001,7.727,148.894
C02527=1135.326,216.339,-65.302,-177.999,7.730,148.894
C02528=1135.322,216.589,-65.327,-177.996,7.733,148.894
C02529=1135.318,216.837,-65.352,-177.993,7.736,148.894
C02530=1135.313,217.085,-65.378,-177.991,7.738,148.894
C02531=1135.309,217.334,-65.403,-177.988,7.741,148.894
C02532=1135.304,217.583,-65.428,-177.985,7.744,148.894
C02533=1135.300,217.832,-65.454,-177.982,7.747,148.893
C02534=1135.296,218.080,-65.480,-177.979,7.749,148.893
C02535=1135.291,218.329,-65.505,-177.976,7.752,148.893
C02536=1135.287,218.577,-65.531,-177.973,7.755,148.893
C02537=1135.282,218.826,-65.557,-177.971,7.757,148.893
C02538=1135.278,219.074,-65.582,-177.968,7.760,148.893
C02539=1135.273,219.323,-65.608,-177.965,7.763,148.893
C02540=1135.269,219.573,-65.633,-177.962,7.766,148.893
C02541=1135.264,219.821,-65.658,-177.960,7.769,148.892
C02542=1135.260,220.069,-65.684,-177.957,7.771,148.892
C02543=1135.255,220.318,-65.710,-177.953,7.774,148.892
C02544=1135.251,220.567,-65.736,-177.951,7.777,148.892
C02545=1135.246,220.815,-65.761,-177.948,7.780,148.892
C02546=1135.241,221.064,-65.787,-177.946,7.782,148.892
C02547=1135.237,221.313,-65.813,-177.943,7.785,148.892
C02548=1135.232,221.561,-65.838,-177.940,7.788,148.891
C02549=1135.228,221.810,-65.864,-177.937,7.791,148.891
C02550=1135.224,222.059,-65.890,-177.934,7.793,148.891
C02551=1135.220,222.308,-65.915,-177.931,7.796,148.891
C02552=1135.214,222.556,-65.941,-177.928,7.799,148.891
C02553=1135.210,222.805,-65.967,-177.925,7.802,148.891
C02554=1135.206,223.053,-65.994,-177.923,7.805,148.891
C02555=1135.202,223.302,-66.019,-177.920,7.808,148.891
C02556=1135.197,223.550,-66.045,-177.918,7.810,148.890
C02557=1135.193,223.799,-66.071,-177.914,7.812,148.890
C02558=1135.188,224.048,-66.097,-177.912,7.815,148.890
C02559=1135.184,224.297,-66.123,-177.909,7.818,148.890
C02560=1135.179,224.545,-66.148,-177.906,7.821,148.890
C02561=1135.175,224.793,-66.175,-177.903,7.824,148.890
C02562=1135.171,225.042,-66.200,-177.900,7.827,148.890
C02563=1135.166,225.291,-66.227,-177.898,7.830,148.890
C02564=1135.161,225.540,-66.252,-177.895,7.833,148.890
C02565=1135.158,225.788,-66.279,-177.892,7.836,148.889
C02566=1135.153,226.036,-66.304,-177.889,7.838,148.889
C02567=1135.148,226.285,-66.331,-177.886,7.841,148.889
C02568=1135.143,226.534,-66.356,-177.883,7.844,148.889
C02569=1135.140,226.782,-66.383,-177.881,7.846,148.889
C02570=1135.135,227.031,-66.409,-177.878,7.849,148.889
C02571=1135.130,227.280,-66.435,-177.875,7.852,148.889
C02572=1135.126,227.527,-66.461,-177.872,7.855,148.889
C02573=1135.121,227.777,-66.487,-177.870,7.858,148.888
C02574=1135.117,228.025,-66.513,-177.867,7.860,148.888
C02575=1135.113,228.274,-66.540,-177.864,7.863,148.888
C02576=1135.108,228.523,-66.566,-177.861,7.866,148.888
C02577=1135.104,228.771,-66.592,-177.858,7.869,148.888
C02578=1135.100,229.020,-66.618,-177.855,7.872,148.888
C02579=1135.095,229.269,-66.644,-177.853,7.875,148.888
C02580=1135.091,229.517,-66.671,-177.850,7.878,148.888
C02581=1135.085,229.765,-66.697,-177.847,7.880,148.888
C02582=1135.081,230.014,-66.723,-177.844,7.883,148.887
C02583=1135.077,230.262,-66.749,-177.841,7.886,148.887
C02584=1135.072,230.511,-66.776,-177.838,7.889,148.887
C02585=1135.068,230.760,-66.802,-177.835,7.892,148.887
C02586=1135.064,231.008,-66.829,-177.833,7.895,148.887
C02587=1135.059,231.257,-66.855,-177.830,7.898,148.887
C02588=1135.055,231.505,-66.882,-177.827,7.901,148.887
C02589=1135.051,231.754,-66.908,-177.825,7.903,148.887
C02590=1135.046,232.003,-66.935,-177.822,7.906,148.887
C02591=1135.042,232.251,-66.961,-177.819,7.909,148.887
C02592=1135.037,232.500,-66.987,-177.816,7.912,148.887
C02593=1135.033,232.748,-67.014,-177.814,7.915,148.886
C02594=1135.028,232.997,-67.041,-177.811,7.917,148.886
C02595=1135.024,233.246,-67.067,-177.808,7.920,148.886
C02596=1135.019,233.494,-67.094,-177.805,7.923,148.886
C02597=1135.016,233.742,-67.120,-177.802,7.926,148.886
C02598=1135.011,233.991,-67.147,-177.799,7.929,148.886
C02599=1135.007,234.240,-67.173,-177.797,7.932,148.886
C02600=1135.002,234.488,-67.200,-177.794,7.935,148.886
C02601=1134.998,234.737,-67.226,-177.791,7.938,148.886
C02602=1134.993,235.008,-67.255,-177.788,7.941,148.886
C02603=1134.987,235.280,-67.285,-177.785,7.944,148.886
C02604=1134.983,235.552,-67.314,-177.782,7.947,148.886
C02605=1134.978,235.825,-67.343,-177.778,7.951,148.885
C02606=1134.974,236.073,-67.369,-177.775,7.954,148.885
C02607=1134.969,236.321,-67.396,-177.773,7.956,148.885
C02608=1134.965,236.569,-67.423,-177.770,7.959,148.885
C02609=1134.960,236.818,-67.450,-177.767,7.962,148.885
C02610=1134.956,237.067,-67.477,-177.764,7.965,148.885
C02611=1134.952,237.316,-67.503,-177.761,7.968,148.885
C02612=1134.947,237.564,-67.530,-177.759,7.971,148.885
C02613=1134.943,237.813,-67.557,-177.756,7.974,148.885
C02614=1134.938,238.061,-67.584,-177.753,7.977,148.885
C02615=1134.934,238.310,-67.611,-177.751,7.980,148.885
C02616=1134.930,238.558,-67.638,-177.748,7.983,148.885
C02617=1134.925,238.807,-67.665,-177.745,7.986,148.884
C02618=1134.921,239.055,-67.691,-177.742,7.989,148.884
C02619=1134.916,239.303,-67.718,-177.739,7.992,148.884
C02620=1134.912,239.552,-67.745,-177.737,7.995,148.884
C02621=1134.908,239.801,-67.773,-177.734,7.998,148.884
C02622=1134.904,240.049,-67.799,-177.731,8.000,148.884
C02623=1134.899,240.298,-67.826,-177.728,8.003,148.884
C02624=1134.894,240.546,-67.854,-177.725,8.006,148.884
C02625=1134.890,240.795,-67.881,-177.723,8.009,148.884
C02626=1134.885,241.043,-67.908,-177.720,8.012,148.884
C02627=1134.882,241.292,-67.934,-177.717,8.015,148.884
C02628=1134.877,241.540,-67.962,-177.714,8.018,148.884
C02629=1134.873,241.788,-67.989,-177.711,8.021,148.884
C02630=1134.852,242.978,-68.120,-178.631,9.818,149.573
C02631=1134.847,243.226,-68.147,-178.629,9.820,149.573
C02632=1134.843,243.474,-68.175,-178.627,9.822,149.573
C02633=1134.839,243.723,-68.203,-178.626,9.825,149.573
C02634=1134.834,243.971,-68.230,-178.625,9.826,149.573
C02635=1134.830,244.219,-68.258,-178.623,9.829,149.573
C02636=1134.826,244.468,-68.286,-178.622,9.831,149.573
C02637=1134.822,244.716,-68.313,-178.621,9.832,149.573
C02638=1134.816,244.965,-68.341,-178.619,9.834,149.573
C02639=1134.812,245.213,-68.369,-178.618,9.836,149.574
C02640=1134.808,245.462,-68.396,-178.617,9.838,149.574
C02641=1134.803,245.710,-68.424,-178.615,9.841,149.574
C02642=1134.799,245.959,-68.451,-178.614,9.843,149.574
C02643=1134.795,246.207,-68.479,-178.614,9.844,149.574
C02644=1134.791,246.455,-68.507,-178.612,9.846,149.574
C02645=1134.787,246.704,-68.534,-178.611,9.848,149.575
C02646=1134.782,246.952,-68.563,-178.611,9.850,149.575
C02647=1134.777,247.201,-68.590,-178.610,9.852,149.575
C02648=1134.773,247.449,-68.618,-178.607,9.855,149.575
C02649=1134.769,247.697,-68.646,-178.599,9.861,149.574
C02650=1134.765,247.946,-68.673,-178.591,9.867,149.574
C02651=1134.760,248.194,-68.701,-178.583,9.874,149.573
C02652=1134.756,248.443,-68.730,-178.575,9.879,149.572
C02653=1134.752,248.691,-68.757,-178.568,9.884,149.572
C02654=1134.747,248.939,-68.785,-178.561,9.889,149.571
C02655=1134.743,249.188,-68.813,-178.555,9.894,149.571
C02656=1134.738,249.436,-68.841,-178.548,9.899,149.570
C02657=1134.734,249.685,-68.869,-178.542,9.903,149.570
C02658=1134.730,249.933,-68.897,-178.537,9.908,149.569
C02659=1134.725,250.182,-68.926,-178.531,9.912,149.569
C02660=1134.721,250.429,-68.954,-178.526,9.916,149.568
C02661=1134.717,250.678,-68.982,-178.521,9.919,149.568
C02662=1134.712,250.926,-69.010,-178.516,9.923,149.567
C02663=1134.709,251.175,-69.038,-178.512,9.926,149.567
C02664=1134.704,251.424,-69.067,-178.508,9.930,149.567
C02665=1134.700,251.672,-69.095,-178.505,9.932,149.567
C02666=1134.695,251.920,-69.123,-178.501,9.935,149.566
C02667=1134.691,252.168,-69.151,-178.499,9.937,149.566
C02668=1134.687,252.417,-69.179,-178.496,9.940,149.566
C02669=1134.682,252.664,-69.208,-178.493,9.942,149.566
C02670=1134.679,252.913,-69.237,-178.491,9.944,149.566
C02671=1134.673,253.236,-69.273,-178.489,9.946,149.566
C02672=1134.667,253.559,-69.310,-178.487,9.948,149.566
C02673=1134.661,253.882,-69.348,-178.486,9.950,149.566
C02674=1134.655,254.205,-69.384,-178.485,9.952,149.566
C02675=1134.652,254.454,-69.413,-178.485,9.953,149.566
C02676=1134.647,254.702,-69.441,-178.485,9.953,149.567
C02677=1134.643,254.950,-69.469,-178.486,9.954,149.567
C02678=1134.639,255.199,-69.499,-178.487,9.954,149.567
C02679=1134.634,255.447,-69.526,-178.487,9.955,149.568
C02680=1134.630,255.695,-69.555,-178.489,9.955,149.568
C02681=1134.626,255.943,-69.583,-178.490,9.955,149.568
C02682=1134.621,256.192,-69.612,-178.488,9.958,149.568
C02683=1134.617,256.441,-69.640,-178.484,9.962,149.568
C02684=1134.612,256.688,-69.669,-178.481,9.964,149.568
C02685=1134.609,256.937,-69.697,-178.478,9.967,149.568
C02686=1134.604,257.185,-69.725,-178.475,9.970,149.568
C02687=1134.600,257.434,-69.754,-178.472,9.973,149.568
C02688=1134.596,257.682,-69.783,-178.469,9.975,149.568
C02689=1134.591,257.930,-69.811,-178.466,9.979,149.568
C02690=1134.587,258.179,-69.839,-178.463,9.982,149.568
C02691=1134.582,258.428,-69.868,-178.460,9.985,149.567
C02692=1134.578,258.675,-69.897,-178.456,9.988,149.567
C02693=1134.574,258.924,-69.925,-178.453,9.991,149.567
C02694=1134.570,259.172,-69.954,-178.449,9.994,149.567
C02695=1134.565,259.420,-69.983,-178.447,9.997,149.567
C02696=1134.561,259.669,-70.011,-178.443,10.000,149.567
C02697=1134.557,259.917,-70.040,-178.440,10.003,149.567
C02698=1134.552,260.165,-70.069,-178.436,10.006,149.566
C02699=1134.548,260.414,-70.097,-178.432,10.010,149.566
C02700=1134.544,260.662,-70.126,-178.429,10.012,149.566
C02701=1134.539,260.910,-70.155,-178.426,10.016,149.566
C02702=1134.535,261.158,-70.184,-178.422,10.019,149.566
C02703=1134.531,261.407,-70.212,-178.418,10.022,149.565
C02704=1134.527,261.655,-70.242,-178.414,10.026,149.565
C02705=1134.522,261.903,-70.270,-178.411,10.028,149.565
C02706=1134.519,262.151,-70.299,-178.407,10.031,149.565
C02707=1134.514,262.400,-70.328,-178.403,10.035,149.565
C02708=1134.510,262.648,-70.357,-178.399,10.038,149.564
C02709=1134.505,262.896,-70.386,-178.395,10.041,149.564
C02710=1134.501,263.145,-70.415,-178.392,10.045,149.564
C02711=1134.497,263.393,-70.444,-178.388,10.048,149.564
C02712=1134.493,263.642,-70.473,-178.384,10.051,149.563
C02713=1134.488,263.889,-70.502,-178.379,10.055,149.563
C02714=1134.484,264.137,-70.531,-178.375,10.058,149.563
C02715=1134.479,264.386,-70.560,-178.371,10.061,149.562
C02716=1134.475,264.635,-70.589,-178.369,10.063,149.562
C02717=1134.472,264.883,-70.618,-178.366,10.066,149.562
C02718=1134.467,265.130,-70.647,-178.363,10.068,149.562
C02719=1134.462,265.379,-70.676,-178.361,10.070,149.562
C02720=1134.458,265.627,-70.705,-178.359,10.073,149.562
C02721=1134.454,265.876,-70.735,-178.356,10.075,149.562
C02722=1134.450,266.124,-70.764,-178.354,10.077,149.562
C02723=1134.446,266.338,-70.789,-178.352,10.079,149.562
C02724=1134.442,266.551,-70.814,-178.350,10.081,149.562
C02725=1134.439,266.766,-70.840,-178.347,10.083,149.562
C02726=1134.435,266.980,-70.865,-178.345,10.085,149.561
C02727=1134.431,267.193,-70.890,-178.343,10.088,149.562
C02728=1134.428,267.408,-70.915,-178.341,10.090,149.561
C02729=1134.424,267.622,-70.940,-178.339,10.092,149.561
C02730=1134.420,267.835,-70.966,-178.336,10.093,149.561
C02731=1134.416,268.083,-70.995,-178.334,10.095,149.561
C02732=1134.412,268.332,-71.024,-178.331,10.099,149.561
C02733=1134.407,268.581,-71.053,-178.329,10.101,149.561
C02734=1134.403,268.829,-71.083,-178.326,10.103,149.561
C02735=1134.399,269.077,-71.112,-178.323,10.106,149.561
C02736=1134.395,269.325,-71.142,-178.321,10.108,149.561
C02737=1134.391,269.574,-71.171,-178.318,10.111,149.561
C02738=1134.386,269.822,-71.200,-178.315,10.114,149.560
C02739=1134.382,270.070,-71.230,-178.313,10.116,149.560
C02740=1134.377,270.318,-71.259,-178.310,10.118,149.560
C02741=1134.373,270.566,-71.288,-178.307,10.121,149.560
C02742=1134.369,270.814,-71.318,-178.304,10.124,149.560
C02743=1134.365,271.063,-71.347,-178.302,10.126,149.560
C02744=1134.361,271.311,-71.377,-178.299,10.129,149.560
C02745=1134.357,271.559,-71.406,-178.296,10.131,149.560
C02746=1134.352,271.807,-71.436,-178.293,10.134,149.560
C02747=1134.348,272.056,-71.465,-178.290,10.137,149.560
C02748=1134.344,272.303,-71.495,-178.287,10.140,149.559
C02749=1134.339,272.552,-71.525,-178.284,10.142,149.559
C02750=1134.335,272.800,-71.555,-178.281,10.145,149.559
C02751=1134.331,273.048,-71.584,-178.278,10.148,149.559
C02752=1134.327,273.297,-71.614,-178.275,10.150,149.559
C02753=1134.323,273.545,-71.643,-178.272,10.153,149.559
C02754=1134.318,273.793,-71.673,-178.269,10.156,149.559
C02755=1134.315,274.041,-71.703,-178.266,10.159,149.559
C02756=1134.310,274.289,-71.733,-178.263,10.161,149.558
C02757=1134.305,274.538,-71.762,-178.260,10.164,149.558
C02758=1134.301,274.786,-71.792,-178.257,10.166,149.558
C02759=1134.297,275.034,-71.822,-178.253,10.169,149.558
C02760=1134.293,275.282,-71.851,-178.250,10.172,149.558
C02761=1134.289,275.530,-71.881,-178.247,10.174,149.558
C02762=1134.284,275.778,-71.912,-178.244,10.178,149.557
C02763=1134.280,276.026,-71.941,-178.241,10.180,149.557
C02764=1134.276,276.275,-71.970,-178.238,10.183,149.557
C02765=1134.272,276.522,-72.001,-178.234,10.186,149.557
C02766=1134.267,276.771,-72.031,-178.231,10.189,149.557
C02767=1134.264,277.020,-72.061,-178.227,10.191,149.556
C02768=1134.260,277.267,-72.091,-178.224,10.194,149.556
C02769=1134.256,277.516,-72.120,-178.220,10.197,149.556
C02770=1134.251,277.764,-72.150,-178.218,10.200,149.556
C02771=1134.247,278.012,-72.180,-178.214,10.203,149.556
C02772=1134.243,278.260,-72.210,-178.211,10.206,149.556
C02773=1134.238,278.508,-72.241,-178.207,10.209,149.555
C02774=1134.234,278.756,-72.270,-178.203,10.212,149.555
C02775=1134.230,279.004,-72.300,-178.200,10.214,149.555
C02776=1134.226,279.253,-72.331,-178.197,10.217,149.555
C02777=1134.222,279.501,-72.361,-178.193,10.220,149.554
C02778=1134.218,279.749,-72.390,-178.190,10.223,149.554
C02779=1134.214,279.962,-72.417,-178.187,10.225,149.554
C02780=1134.210,280.177,-72.443,-178.184,10.228,149.554
C02781=1134.206,280.390,-72.468,-178.180,10.230,149.554
C02782=1134.203,280.604,-72.495,-178.177,10.233,149.553
C02783=1134.199,280.819,-72.521,-178.174,10.236,149.553
C02784=1134.195,281.032,-72.547,-178.171,10.238,149.553
C02785=1134.192,281.246,-72.573,-178.168,10.241,149.553
C02786=1134.188,281.459,-72.599,-178.165,10.243,149.553
C02787=1134.185,281.708,-72.629,-178.162,10.246,149.552
C02788=1134.180,281.956,-72.659,-178.158,10.248,149.552
C02789=1134.176,282.204,-72.690,-178.155,10.251,149.552
C02790=1134.171,282.452,-72.720,-178.152,10.254,149.552
C02791=1134.167,282.700,-72.751,-178.149,10.256,149.552
C02792=1134.163,282.949,-72.781,-178.146,10.259,149.552
C02793=1134.159,283.197,-72.811,-178.143,10.261,149.551
C02794=1134.155,283.445,-72.842,-178.140,10.263,149.551
C02795=1134.150,283.693,-72.873,-178.137,10.266,149.551
C02796=1134.146,283.941,-72.902,-178.134,10.269,149.551
C02797=1134.142,284.189,-72.933,-178.131,10.271,149.551
C02798=1134.138,284.437,-72.963,-178.128,10.274,149.550
C02799=1134.133,284.685,-72.994,-178.125,10.277,149.550
C02800=1134.129,284.933,-73.024,-178.122,10.279,149.550
C02801=1134.125,285.181,-73.055,-178.119,10.282,149.550
C02802=1134.121,285.430,-73.086,-178.115,10.284,149.550
C02803=1134.117,285.678,-73.116,-178.112,10.287,149.550
C02804=1134.113,285.926,-73.147,-178.110,10.289,149.549
C02805=1134.109,286.174,-73.177,-178.107,10.291,149.549
C02806=1134.104,286.422,-73.208,-178.103,10.294,149.549
C02807=1134.100,286.670,-73.239,-178.100,10.297,149.549
C02808=1134.096,286.918,-73.269,-178.098,10.299,149.549
C02809=1134.092,287.166,-73.300,-178.094,10.302,149.548
C02810=1134.087,287.414,-73.331,-178.091,10.304,149.548
C02811=1134.084,287.662,-73.361,-178.088,10.307,149.548
C02812=1134.079,287.910,-73.392,-178.085,10.310,149.548
C02813=1134.075,288.158,-73.423,-178.082,10.312,149.548
C02814=1134.071,288.407,-73.453,-178.079,10.315,149.548
C02815=1134.067,288.655,-73.484,-178.076,10.316,149.547
C02816=1134.062,288.903,-73.515,-178.073,10.319,149.547
C02817=1134.059,289.151,-73.545,-178.070,10.322,149.547
C02818=1134.054,289.398,-73.577,-178.067,10.324,149.547
C02819=1134.050,289.646,-73.608,-178.064,10.327,149.547
C02820=1134.046,289.895,-73.639,-178.060,10.330,149.546
C02821=1134.042,290.143,-73.669,-178.058,10.332,149.546
C02822=1134.038,290.391,-73.700,-178.054,10.335,149.546
C02823=1134.033,290.639,-73.731,-178.051,10.338,149.546
C02824=1134.029,290.887,-73.761,-178.048,10.340,149.546
C02825=1134.025,291.135,-73.793,-178.045,10.343,149.546
C02826=1134.021,291.383,-73.823,-178.042,10.345,149.545
C02827=1134.017,291.631,-73.855,-178.039,10.348,149.545
C02828=1134.013,291.879,-73.885,-178.036,10.350,149.545
C02829=1134.008,292.127,-73.917,-178.033,10.352,149.545
C02830=1134.004,292.375,-73.948,-178.030,10.355,149.545
C02831=1134.000,292.623,-73.978,-178.027,10.357,149.545
C02832=1133.997,292.871,-74.010,-178.023,10.360,149.544
C02833=1133.992,293.119,-74.041,-178.021,10.363,149.544
C02834=1133.988,293.368,-74.072,-178.017,10.365,149.544
C02835=1133.984,293.581,-74.098,-178.015,10.367,149.544
C02836=1133.981,293.795,-74.125,-178.012,10.370,149.544
C02837=1133.977,294.008,-74.152,-178.010,10.372,149.544
C02838=1133.974,294.222,-74.179,-178.007,10.373,149.543
C02839=1133.970,294.436,-74.206,-178.004,10.376,149.543
C02840=1133.966,294.649,-74.232,-178.002,10.378,149.543
C02841=1133.962,294.863,-74.260,-177.998,10.381,149.543
C02842=1133.959,295.077,-74.287,-177.996,10.383,149.543
C02843=1133.955,295.325,-74.318,-177.993,10.385,149.543
C02844=1133.951,295.573,-74.349,-177.990,10.388,149.542
C02845=1133.948,295.821,-74.380,-177.987,10.391,149.542
C02846=1133.943,296.069,-74.411,-177.984,10.393,149.542
C02847=1133.939,296.317,-74.443,-177.981,10.396,149.542
C02848=1133.935,296.565,-74.474,-177.977,10.398,149.542
C02849=1133.931,296.813,-74.506,-177.974,10.401,149.542
C02850=1133.926,297.061,-74.536,-177.972,10.403,149.541
C02851=1133.923,297.309,-74.568,-177.969,10.405,149.541
C02852=1133.918,297.557,-74.599,-177.965,10.408,149.541
C02853=1133.914,297.805,-74.632,-177.962,10.411,149.541
C02854=1133.909,298.053,-74.663,-177.959,10.413,149.541
C02855=1133.905,298.301,-74.694,-177.956,10.416,149.540
C02856=1133.901,298.549,-74.726,-177.953,10.418,149.540
C02857=1133.897,298.797,-74.757,-177.950,10.421,149.540
C02858=1133.893,299.045,-74.788,-177.947,10.423,149.540
C02859=1133.889,299.293,-74.820,-177.944,10.426,149.540
C02860=1133.885,299.541,-74.851,-177.940,10.429,149.539
C02861=1133.881,299.789,-74.883,-177.937,10.431,149.539
C02862=1133.877,300.037,-74.915,-177.934,10.434,149.539
C02863=1133.873,300.284,-74.946,-177.931,10.437,149.539
C02864=1133.869,300.533,-74.977,-177.928,10.438,149.539
C02865=1133.864,300.781,-75.010,-177.925,10.441,149.539
C02866=1133.860,301.028,-75.041,-177.922,10.443,149.538
C02867=1133.856,301.276,-75.073,-177.919,10.446,149.538
C02868=1133.851,301.524,-75.104,-177.916,10.449,149.538
C02869=1133.848,301.772,-75.135,-177.912,10.451,149.538
C02870=1133.843,302.021,-75.168,-177.910,10.454,149.538
C02871=1133.839,302.268,-75.199,-177.906,10.456,149.537
C02872=1133.835,302.516,-75.231,-177.903,10.459,149.537
C02873=1133.832,302.764,-75.263,-177.900,10.461,149.537
C02874=1133.827,303.012,-75.294,-177.897,10.464,149.537
C02875=1133.823,303.260,-75.326,-177.894,10.467,149.537
C02876=1133.818,303.508,-75.358,-177.891,10.469,149.537
C02877=1133.815,303.756,-75.390,-177.887,10.472,149.536
C02878=1133.811,304.004,-75.421,-177.884,10.475,149.536
C02879=1133.806,304.251,-75.454,-177.881,10.477,149.536
C02880=1133.802,304.499,-75.485,-177.878,10.479,149.536
C02881=1133.798,304.748,-75.517,-177.876,10.481,149.536
C02882=1133.794,304.996,-75.550,-177.872,10.484,149.535
C02883=1133.790,305.243,-75.581,-177.869,10.487,149.535
C02884=1133.786,305.491,-75.613,-177.866,10.489,149.535
C02885=1133.781,305.740,-75.645,-177.863,10.492,149.535
C02886=1133.777,305.987,-75.677,-177.860,10.494,149.535
C02887=1133.773,306.235,-75.709,-177.857,10.497,149.535
C02888=1133.769,306.483,-75.741,-177.853,10.499,149.534
C02889=1133.765,306.731,-75.773,-177.850,10.502,149.534
C02890=1133.761,306.979,-75.805,-177.847,10.505,149.534
C02891=1133.757,307.192,-75.833,-177.845,10.507,149.534
C02892=1133.754,307.405,-75.860,-177.841,10.509,149.534
C02893=1133.750,307.620,-75.888,-177.839,10.511,149.534
C02894=1133.747,307.833,-75.915,-177.837,10.513,149.533
C02895=1133.743,308.046,-75.943,-177.834,10.516,149.533
C02896=1133.740,308.259,-75.971,-177.831,10.517,149.533
C02897=1133.736,308.474,-75.998,-177.828,10.520,149.533
C02898=1133.733,308.687,-76.026,-177.826,10.522,149.533
C02899=1133.728,308.935,-76.059,-177.823,10.525,149.533
C02900=1133.725,309.183,-76.091,-177.819,10.527,149.532
C02901=1133.720,309.431,-76.124,-177.816,10.530,149.532
C02902=1133.717,309.679,-76.155,-177.813,10.532,149.532
C02903=1133.712,309.927,-76.187,-177.810,10.535,149.532
C02904=1133.708,310.174,-76.220,-177.807,10.538,149.532
C02905=1133.704,310.422,-76.252,-177.804,10.540,149.531
C02906=1133.700,310.670,-76.284,-177.800,10.542,149.531
C02907=1133.696,310.918,-76.317,-177.797,10.545,149.531
C02908=1133.692,311.165,-76.349,-177.794,10.548,149.531
C02909=1133.687,311.414,-76.381,-177.792,10.550,149.531
C02910=1133.684,311.661,-76.414,-177.788,10.552,149.530
C02911=1133.679,311.910,-76.446,-177.785,10.555,149.530
C02912=1133.676,312.158,-76.478,-177.782,10.557,149.530
C02913=1133.672,312.405,-76.511,-177.779,10.560,149.530
C02914=1133.668,312.653,-76.543,-177.776,10.562,149.530
C02915=1133.663,312.900,-76.576,-177.772,10.565,149.530
C02916=1133.659,313.149,-76.608,-177.770,10.568,149.529
C02917=1133.655,313.396,-76.641,-177.766,10.570,149.529
C02918=1133.651,313.645,-76.673,-177.763,10.573,149.529
C02919=1133.647,313.892,-76.706,-177.760,10.575,149.529
C02920=1133.643,314.140,-76.738,-177.757,10.578,149.529
C02921=1133.639,314.388,-76.772,-177.753,10.580,149.528
C02922=1133.635,314.636,-76.803,-177.750,10.583,149.528
C02923=1133.631,314.884,-76.837,-177.747,10.585,149.528
C02924=1133.627,315.132,-76.868,-177.744,10.588,149.528
C02925=1133.623,315.379,-76.901,-177.741,10.591,149.528
C02926=1133.618,315.627,-76.934,-177.737,10.593,149.527
C02927=1133.615,315.875,-76.966,-177.735,10.596,149.527
C02928=1133.611,316.122,-76.999,-177.731,10.598,149.527
C02929=1133.606,316.371,-77.032,-177.729,10.600,149.527
C02930=1133.602,316.618,-77.065,-177.726,10.603,149.527
C02931=1133.599,316.866,-77.098,-177.722,10.605,149.527
C02932=1133.594,317.114,-77.130,-177.719,10.608,149.526
C02933=1133.590,317.362,-77.163,-177.716,10.610,149.526
C02934=1133.587,317.609,-77.196,-177.713,10.613,149.526
C02935=1133.582,317.857,-77.229,-177.710,10.616,149.526
C02936=1133.578,318.105,-77.261,-177.706,10.618,149.526
C02937=1133.574,318.353,-77.294,-177.703,10.620,149.525
C02938=1133.570,318.601,-77.327,-177.700,10.623,149.525
C02939=1133.566,318.848,-77.360,-177.697,10.626,149.525
C02940=1133.562,319.096,-77.393,-177.694,10.628,149.525
C02941=1133.558,319.344,-77.426,-177.691,10.631,149.525
C02942=1133.554,319.592,-77.459,-177.687,10.633,149.524
C02943=1133.550,319.840,-77.491,-177.684,10.636,149.524
C02944=1133.546,320.087,-77.525,-177.681,10.639,149.524
C02945=1133.542,320.335,-77.558,-177.678,10.641,149.524
C02946=1133.538,320.583,-77.591,-177.675,10.644,149.524
C02947=1133.534,320.796,-77.619,-177.672,10.645,149.524
C02948=1133.531,321.010,-77.648,-177.669,10.648,149.523
C02949=1133.528,321.223,-77.676,-177.666,10.650,149.523
C02950=1133.524,321.437,-77.704,-177.664,10.652,149.523
C02951=1133.521,321.649,-77.733,-177.661,10.654,149.523
C02952=1133.517,321.864,-77.762,-177.658,10.656,149.523
C02953=1133.514,322.077,-77.790,-177.656,10.659,149.523
C02954=1133.510,322.290,-77.819,-177.653,10.661,149.522
C02955=1133.506,322.538,-77.852,-177.650,10.663,149.522
C02956=1133.502,322.785,-77.885,-177.647,10.666,149.522
C02957=1133.498,323.034,-77.918,-177.643,10.668,149.522
C02958=1133.494,323.282,-77.952,-177.640,10.671,149.522
C02959=1133.491,323.529,-77.984,-177.637,10.674,149.522
C02960=1133.487,323.777,-78.017,-177.634,10.676,149.521
C02961=1133.482,324.025,-78.050,-177.630,10.678,149.521
C02962=1133.478,324.272,-78.084,-177.627,10.681,149.521
C02963=1133.474,324.520,-78.117,-177.624,10.684,149.521
C02964=1133.470,324.767,-78.151,-177.621,10.686,149.520
C02965=1133.467,325.016,-78.184,-177.618,10.689,149.520
C02966=1133.463,325.263,-78.217,-177.615,10.691,149.520
C02967=1133.458,325.511,-78.250,-177.611,10.694,149.520
C02968=1133.454,325.759,-78.284,-177.609,10.696,149.520
C02969=1133.449,326.007,-78.317,-177.606,10.698,149.520
C02970=1133.446,326.254,-78.351,-177.602,10.701,149.519
C02971=1133.442,326.502,-78.384,-177.599,10.703,149.519
C02972=1133.438,326.750,-78.418,-177.596,10.706,149.519
C02973=1133.434,326.998,-78.451,-177.593,10.708,149.519
C02974=1133.430,327.245,-78.485,-177.589,10.711,149.519
C02975=1133.426,327.493,-78.518,-177.586,10.714,149.518
C02976=1133.422,327.740,-78.551,-177.583,10.716,149.518
C02977=1133.418,327.988,-78.585,-177.580,10.718,149.518
C02978=1133.414,328.236,-78.619,-177.577,10.721,149.518
C02979=1133.410,328.484,-78.652,-177.574,10.724,149.518
C02980=1133.406,328.731,-78.686,-177.570,10.726,149.517
C02981=1133.402,328.979,-78.719,-177.567,10.729,149.517
C02982=1133.398,329.227,-78.753,-177.564,10.731,149.517
C02983=1133.394,329.474,-78.787,-177.561,10.734,149.517
C02984=1133.390,329.722,-78.820,-177.557,10.736,149.517
C02985=1133.386,329.969,-78.854,-177.554,10.739,149.516
C02986=1133.382,330.218,-78.888,-177.551,10.741,149.516
C02987=1133.378,330.465,-78.922,-177.548,10.744,149.516
C02988=1133.374,330.713,-78.955,-177.545,10.746,149.516
C02989=1133.370,330.960,-78.989,-177.542,10.749,149.516
C02990=1133.366,331.209,-79.023,-177.538,10.752,149.516
C02991=1133.362,331.456,-79.057,-177.535,10.754,149.515
C02992=1133.358,331.703,-79.090,-177.532,10.756,149.515
C02993=1133.355,331.951,-79.124,-177.529,10.759,149.515
C02994=1133.350,332.199,-79.158,-177.525,10.762,149.515
C02995=1133.346,332.446,-79.192,-177.522,10.764,149.514
C02996=1133.342,332.694,-79.225,-177.519,10.767,149.514
C02997=1133.339,332.942,-79.259,-177.516,10.769,149.514
C02998=1133.334,333.189,-79.294,-177.513,10.771,149.514
C02999=1133.330,333.437,-79.327,-177.510,10.774,149.514
C03000=1133.327,333.685,-79.361,-177.506,10.776,149.513
C03001=1133.322,333.932,-79.396,-177.504,10.779,149.513
C03002=1133.318,334.180,-79.429,-177.500,10.781,149.513
C03003=1133.315,334.394,-79.458,-177.497,10.784,149.513
C03004=1133.311,334.607,-79.487,-177.495,10.786,149.513
C03005=1133.308,334.820,-79.517,-177.491,10.788,149.513
C03006=1133.305,335.033,-79.546,-177.489,10.790,149.512
C03007=1133.302,335.246,-79.576,-177.486,10.792,149.512
C03008=1133.297,335.459,-79.605,-177.483,10.795,149.512
C03009=1133.294,335.673,-79.634,-177.481,10.796,149.512
C03010=1133.291,335.886,-79.663,-177.478,10.799,149.512
C03011=1133.287,336.134,-79.698,-177.474,10.801,149.512
C03012=1133.283,336.381,-79.732,-177.471,10.804,149.511
C03013=1133.278,336.629,-79.766,-177.468,10.806,149.511
C03014=1133.275,336.877,-79.800,-177.465,10.809,149.511
C03015=1133.271,337.124,-79.834,-177.462,10.812,149.511
C03016=1133.267,337.372,-79.869,-177.458,10.814,149.511
C03017=1133.263,337.619,-79.902,-177.455,10.816,149.510
C03018=1133.259,337.867,-79.937,-177.452,10.818,149.510
C03019=1133.256,338.115,-79.971,-177.449,10.821,149.510
C03020=1133.251,338.362,-80.006,-177.446,10.823,149.510
C03021=1133.248,338.610,-80.040,-177.443,10.826,149.510
C03022=1133.243,338.857,-80.074,-177.439,10.828,149.509
C03023=1133.240,339.106,-80.108,-177.436,10.831,149.509
C03024=1133.235,339.353,-80.142,-177.433,10.833,149.509
C03025=1133.231,339.600,-80.176,-177.430,10.836,149.509
C03026=1133.227,339.848,-80.211,-177.427,10.838,149.509
C03027=1133.223,340.096,-80.245,-177.423,10.841,149.508
C03028=1133.220,340.343,-80.280,-177.420,10.843,149.508
C03029=1133.215,340.590,-80.315,-177.417,10.846,149.508
C03030=1133.212,340.838,-80.349,-177.414,10.849,149.508
C03031=1133.207,341.085,-80.384,-177.410,10.851,149.508
C03032=1133.203,341.334,-80.418,-177.407,10.854,149.507
C03033=1133.200,341.581,-80.452,-177.404,10.856,149.507
C03034=1133.196,341.829,-80.487,-177.400,10.858,149.507
C03035=1133.192,342.076,-80.521,-177.397,10.861,149.507
C03036=1133.188,342.324,-80.556,-177.394,10.864,149.507
C03037=1133.183,342.572,-80.590,-177.391,10.866,149.506
C03038=1133.180,342.819,-80.625,-177.388,10.869,149.506
C03039=1133.176,343.066,-80.660,-177.384,10.871,149.506
C03040=1133.172,343.314,-80.695,-177.381,10.873,149.506
C03041=1133.168,343.561,-80.728,-177.378,10.876,149.505
C03042=1133.164,343.809,-80.763,-177.375,10.879,149.505
C03043=1133.160,344.056,-80.798,-177.371,10.881,149.505
C03044=1133.156,344.304,-80.833,-177.368,10.884,149.505
C03045=1133.152,344.551,-80.867,-177.365,10.886,149.505
C03046=1133.148,344.799,-80.903,-177.361,10.889,149.504
C03047=1133.144,345.047,-80.938,-177.358,10.891,149.504
C03048=1133.141,345.294,-80.971,-177.355,10.893,149.504
C03049=1133.137,345.542,-81.007,-177.352,10.896,149.504
C03050=1133.132,345.789,-81.041,-177.349,10.899,149.504
C03051=1133.128,346.037,-81.076,-177.345,10.901,149.503
C03052=1133.124,346.284,-81.111,-177.342,10.904,149.503
C03053=1133.121,346.532,-81.146,-177.339,10.906,149.503
C03054=1133.117,346.780,-81.180,-177.335,10.909,149.503
C03055=1133.113,347.027,-81.216,-177.332,10.911,149.503
C03056=1133.109,347.275,-81.251,-177.329,10.913,149.502
C03057=1133.105,347.522,-81.286,-177.326,10.916,149.502
C03058=1133.101,347.770,-81.320,-177.322,10.919,149.502
C03059=1133.098,347.983,-81.350,-177.320,10.920,149.502
C03060=1133.094,348.196,-81.381,-177.317,10.922,149.501
C03061=1133.090,348.409,-81.411,-177.314,10.925,149.501
C03062=1133.088,348.622,-81.440,-177.311,10.927,149.501
C03063=1133.084,348.836,-81.471,-177.309,10.929,149.501
C03064=1133.080,349.048,-81.501,-177.306,10.931,149.501
C03065=1133.078,349.261,-81.531,-177.303,10.933,149.501
C03066=1133.074,349.474,-81.562,-177.300,10.935,149.501
C03067=1133.070,349.722,-81.596,-177.297,10.938,149.500
C03068=1133.066,349.969,-81.632,-177.293,10.941,149.500
C03069=1133.062,350.217,-81.667,-177.289,10.943,149.500
C03070=1133.058,350.465,-81.702,-177.285,10.946,149.499
C03071=1133.054,350.712,-81.737,-177.282,10.949,149.499
C03072=1133.050,350.959,-81.773,-177.278,10.952,149.499
C03073=1133.047,351.207,-81.808,-177.274,10.954,149.499
C03074=1133.042,351.454,-81.843,-177.270,10.957,149.498
C03075=1133.039,351.702,-81.878,-177.267,10.960,149.498
C03076=1133.035,351.950,-81.913,-177.263,10.962,149.498
C03077=1133.031,352.197,-81.949,-177.259,10.965,149.498
C03078=1133.027,352.444,-81.984,-177.256,10.968,149.497
C03079=1133.023,352.692,-82.020,-177.252,10.971,149.497
C03080=1133.019,352.939,-82.055,-177.248,10.973,149.497
C03081=1133.015,353.187,-82.090,-177.245,10.975,149.496
C03082=1133.011,353.434,-82.125,-177.241,10.979,149.496
C03083=1133.007,353.681,-82.161,-177.238,10.981,149.496
C03084=1133.004,353.929,-82.196,-177.234,10.983,149.496
C03085=1133.000,354.176,-82.232,-177.231,10.986,149.495
C03086=1132.996,354.424,-82.267,-177.227,10.989,149.495
C03087=1132.992,354.671,-82.303,-177.223,10.991,149.495
C03088=1132.989,354.918,-82.338,-177.220,10.994,149.495
C03089=1132.985,355.166,-82.373,-177.216,10.997,149.494
C03090=1132.981,355.414,-82.408,-177.212,10.999,149.494
C03091=1132.977,355.661,-82.444,-177.209,11.001,149.494
C03092=1132.972,355.908,-82.480,-177.205,11.004,149.494
C03093=1132.969,356.156,-82.515,-177.201,11.007,149.493
C03094=1132.965,356.403,-82.551,-177.198,11.009,149.493
C03095=1132.962,356.650,-82.587,-177.194,11.012,149.493
C03096=1132.958,356.898,-82.623,-177.191,11.014,149.493
C03097=1132.954,357.145,-82.658,-177.187,11.016,149.492
C03098=1132.950,357.393,-82.694,-177.184,11.019,149.492
C03099=1132.946,357.640,-82.730,-177.180,11.022,149.492
C03100=1132.942,357.887,-82.765,-177.176,11.024,149.491
C03101=1132.938,358.135,-82.801,-177.173,11.027,149.491
C03102=1132.935,358.382,-82.836,-177.170,11.029,149.491
C03103=1132.930,358.630,-82.872,-177.167,11.032,149.491
C03104=1132.927,358.877,-82.909,-177.163,11.034,149.490
C03105=1132.923,359.125,-82.944,-177.160,11.036,149.490
C03106=1132.920,359.372,-82.980,-177.156,11.039,149.490
C03107=1132.915,359.620,-83.016,-177.153,11.041,149.490
C03108=1132.912,359.867,-83.052,-177.149,11.044,149.489
C03109=1132.908,360.114,-83.088,-177.145,11.046,149.489
C03110=1132.903,360.361,-83.123,-177.142,11.049,149.489
C03111=1132.899,360.609,-83.159,-177.138,11.051,149.488
C03112=1132.896,360.856,-83.195,-177.135,11.054,149.488
C03113=1132.892,361.104,-83.231,-177.132,11.056,149.488
C03114=1132.888,361.351,-83.267,-177.128,11.058,149.488
C03115=1132.885,361.564,-83.298,-177.126,11.060,149.487
C03116=1132.882,361.777,-83.329,-177.122,11.063,149.487
C03117=1132.879,361.990,-83.360,-177.120,11.064,149.487
C03118=1132.876,362.202,-83.391,-177.117,11.066,149.487
C03119=1132.872,362.416,-83.422,-177.114,11.068,149.487
C03120=1132.868,362.629,-83.454,-177.111,11.070,149.486
C03121=1132.865,362.842,-83.484,-177.108,11.073,149.486
C03122=1132.862,363.055,-83.516,-177.105,11.075,149.486
C03123=1132.858,363.302,-83.551,-177.102,11.077,149.486
C03124=1132.854,363.549,-83.588,-177.098,11.079,149.485
C03125=1132.851,363.797,-83.624,-177.095,11.082,149.485
C03126=1132.847,364.044,-83.660,-177.092,11.084,149.485
C03127=1132.843,364.291,-83.696,-177.089,11.087,149.485
C03128=1132.839,364.538,-83.732,-177.085,11.089,149.485
C03129=1132.835,364.786,-83.768,-177.082,11.091,149.484
C03130=1132.832,365.033,-83.805,-177.079,11.093,149.484
C03131=1132.828,365.280,-83.841,-177.076,11.095,149.484
C03132=1132.824,365.528,-83.877,-177.072,11.098,149.483
C03133=1132.820,365.775,-83.914,-177.069,11.100,149.483
C03134=1132.816,366.022,-83.949,-177.066,11.103,149.483
C03135=1132.812,366.270,-83.986,-177.062,11.105,149.483
C03136=1132.809,366.517,-84.023,-177.059,11.108,149.483
C03137=1132.805,366.765,-84.059,-177.056,11.109,149.482
C03138=1132.802,367.012,-84.095,-177.053,11.112,149.482
C03139=1132.797,367.259,-84.132,-177.049,11.114,149.482
C03140=1132.794,367.507,-84.168,-177.046,11.117,149.482
C03141=1132.790,367.754,-84.205,-177.043,11.119,149.481
C03142=1132.786,368.001,-84.241,-177.040,11.121,149.481
C03143=1132.782,368.248,-84.277,-177.037,11.123,149.481
C03144=1132.778,368.496,-84.314,-177.033,11.126,149.481
C03145=1132.775,368.743,-84.350,-177.030,11.128,149.480
C03146=1132.771,368.990,-84.387,-177.027,11.130,149.480
C03147=1132.767,369.238,-84.424,-177.024,11.132,149.480
C03148=1132.763,369.485,-84.460,-177.021,11.135,149.480
C03149=1132.759,369.732,-84.497,-177.018,11.137,149.480
C03150=1132.755,369.979,-84.533,-177.015,11.139,149.479
C03151=1132.752,370.226,-84.570,-177.012,11.142,149.479
C03152=1132.748,370.474,-84.607,-177.009,11.144,149.479
C03153=1132.744,370.721,-84.643,-177.006,11.146,149.479
C03154=1132.741,370.968,-84.680,-177.003,11.148,149.479
C03155=1132.736,371.216,-84.716,-176.999,11.151,149.478
C03156=1132.732,371.463,-84.753,-176.997,11.153,149.478
C03157=1132.729,371.710,-84.789,-176.993,11.155,149.478
C03158=1132.725,371.957,-84.826,-176.990,11.158,149.478
C03159=1132.721,372.205,-84.863,-176.988,11.160,149.478
C03160=1132.718,372.452,-84.900,-176.985,11.162,149.477
C03161=1132.714,372.699,-84.937,-176.981,11.165,149.477
C03162=1132.710,372.947,-84.973,-176.979,11.166,149.477
C03163=1132.706,373.194,-85.010,-176.975,11.169,149.477
C03164=1132.703,373.441,-85.047,-176.972,11.172,149.477
C03165=1132.699,373.689,-85.084,-176.970,11.173,149.477
C03166=1132.695,373.936,-85.121,-176.966,11.176,149.476
C03167=1132.691,374.183,-85.157,-176.963,11.178,149.476
C03168=1132.687,374.430,-85.194,-176.961,11.180,149.476
C03169=1132.684,374.677,-85.232,-176.958,11.183,149.476
C03170=1132.680,374.924,-85.269,-176.955,11.184,149.476
C03171=1132.676,375.137,-85.300,-176.953,11.186,149.476
C03172=1132.673,375.350,-85.332,-176.950,11.188,149.476
C03173=1132.669,375.563,-85.364,-176.947,11.191,149.475
C03174=1132.667,375.776,-85.396,-176.945,11.193,149.475
C03175=1132.663,375.989,-85.428,-176.942,11.195,149.475
C03176=1132.660,376.201,-85.459,-176.940,11.197,149.475
C03177=1132.657,376.414,-85.491,-176.938,11.199,149.475
C03178=1132.654,376.626,-85.523,-176.935,11.200,149.475
C03179=1132.650,376.874,-85.560,-176.933,11.202,149.475
C03180=1132.646,377.121,-85.597,-176.929,11.205,149.474
C03181=1132.642,377.368,-85.634,-176.927,11.207,149.474
C03182=1132.638,377.615,-85.671,-176.924,11.209,149.474
C03183=1132.635,377.863,-85.709,-176.921,11.211,149.474
C03184=1132.631,378.110,-85.745,-176.918,11.214,149.474
C03185=1132.628,378.357,-85.782,-176.915,11.217,149.474
C03186=1132.624,378.604,-85.820,-176.913,11.219,149.474
C03187=1132.620,378.851,-85.857,-176.910,11.221,149.474
C03188=1132.616,379.099,-85.893,-176.907,11.223,149.474
C03189=1132.613,379.346,-85.931,-176.905,11.225,149.473
C03190=1132.609,379.593,-85.968,-176.902,11.228,149.473
C03191=1132.605,379.840,-86.005,-176.900,11.230,149.473
C03192=1132.602,380.088,-86.043,-176.896,11.232,149.473
C03193=1132.597,380.335,-86.080,-176.894,11.234,149.473
C03194=1132.594,380.581,-86.117,-176.891,11.237,149.473
C03195=1132.590,380.829,-86.155,-176.889,11.239,149.473
C03196=1132.586,381.076,-86.192,-176.886,11.242,149.473
C03197=1132.582,381.323,-86.229,-176.883,11.244,149.473
C03198=1132.579,381.571,-86.266,-176.880,11.246,149.473
C03199=1132.575,381.817,-86.304,-176.878,11.248,149.473
C03200=1132.571,382.065,-86.341,-176.876,11.251,149.473
C03201=1132.568,382.312,-86.379,-176.873,11.253,149.473
C03202=1132.564,382.559,-86.416,-176.870,11.255,149.472
C03203=1132.560,382.806,-86.453,-176.867,11.258,149.472
C03204=1132.556,383.054,-86.490,-176.865,11.260,149.472
C03205=1132.553,383.300,-86.528,-176.862,11.263,149.472
C03206=1132.549,383.548,-86.565,-176.861,11.264,149.472
C03207=1132.545,383.795,-86.603,-176.860,11.266,149.472
C03208=1132.541,384.043,-86.641,-176.858,11.267,149.472
C03209=1132.537,384.289,-86.678,-176.857,11.269,149.473
C03210=1132.533,384.536,-86.716,-176.856,11.271,149.473
C03211=1132.530,384.784,-86.753,-176.855,11.272,149.473
C03212=1132.526,385.030,-86.790,-176.854,11.274,149.473
C03213=1132.523,385.278,-86.828,-176.853,11.276,149.473
C03214=1132.519,385.525,-86.865,-176.852,11.278,149.473
C03215=1132.515,385.771,-86.903,-176.851,11.279,149.473
C03216=1132.512,386.019,-86.940,-176.849,11.281,149.474
C03217=1132.508,386.266,-86.978,-176.848,11.283,149.474
C03218=1132.504,386.514,-87.015,-176.848,11.284,149.474
C03219=1132.500,386.761,-87.053,-176.846,11.286,149.474
C03220=1132.497,387.008,-87.091,-176.845,11.288,149.474
C03221=1132.493,387.255,-87.128,-176.844,11.289,149.475
C03222=1132.489,387.502,-87.165,-176.843,11.291,149.475
C03223=1132.486,387.749,-87.203,-176.843,11.293,149.475
C03224=1132.481,387.996,-87.240,-176.842,11.295,149.475
C03225=1132.478,388.243,-87.278,-176.841,11.296,149.476
C03226=1132.474,388.490,-87.316,-176.841,11.298,149.476
C03227=1132.471,388.704,-87.348,-176.839,11.300,149.476
C03228=1132.468,388.916,-87.381,-176.838,11.302,149.476
C03229=1132.464,389.128,-87.413,-176.838,11.304,149.477
C03230=1132.462,389.341,-87.446,-176.837,11.305,149.477
C03231=1132.458,389.554,-87.477,-176.837,11.307,149.477
C03232=1132.455,389.766,-87.510,-176.836,11.309,149.477
C03233=1132.451,389.979,-87.543,-176.835,11.310,149.478
C03234=1132.449,390.192,-87.575,-176.835,11.312,149.478
C03235=1132.445,390.439,-87.612,-176.834,11.313,149.478
C03236=1132.441,390.686,-87.650,-176.833,11.316,149.479
C03237=1132.438,390.933,-87.688,-176.832,11.318,149.479
C03238=1132.434,391.180,-87.726,-176.832,11.320,149.479
C03239=1132.430,391.428,-87.763,-176.831,11.322,149.480
C03240=1132.426,391.675,-87.801,-176.831,11.324,149.480
C03241=1132.423,391.921,-87.839,-176.830,11.326,149.480
C03242=1132.419,392.169,-87.877,-176.829,11.328,149.481
C03243=1132.415,392.416,-87.914,-176.829,11.330,149.481
C03244=1132.412,392.663,-87.952,-176.828,11.332,149.481
C03245=1132.408,392.910,-87.990,-176.828,11.334,149.482
C03246=1132.404,393.157,-88.028,-176.827,11.337,149.482
C03247=1132.401,393.404,-88.065,-176.827,11.339,149.483
C03248=1132.397,393.652,-88.102,-176.826,11.341,149.483
C03249=1132.393,393.899,-88.141,-176.826,11.343,149.484
C03250=1132.389,394.146,-88.179,-176.825,11.346,149.484
C03251=1132.386,394.392,-88.216,-176.825,11.348,149.485
C03252=1132.382,394.640,-88.254,-176.824,11.350,149.485
C03253=1132.378,394.887,-88.291,-176.824,11.352,149.486
C03254=1132.374,395.134,-88.329,-176.824,11.355,149.486
C03255=1132.371,395.381,-88.367,-176.823,11.358,149.487
C03256=1132.367,395.628,-88.405,-176.822,11.360,149.487
C03257=1132.363,395.875,-88.443,-176.822,11.363,149.488
C03258=1132.360,396.123,-88.481,-176.822,11.365,149.488
C03259=1132.356,396.370,-88.518,-176.822,11.367,149.489
C03260=1132.352,396.617,-88.556,-176.821,11.370,149.489
C03261=1132.348,396.864,-88.594,-176.821,11.372,149.490
C03262=1132.345,397.111,-88.632,-176.821,11.375,149.491
C03263=1132.341,397.358,-88.670,-176.821,11.377,149.491
C03264=1132.338,397.605,-88.707,-176.820,11.380,149.492
C03265=1132.333,397.852,-88.746,-176.820,11.382,149.492
C03266=1132.330,398.099,-88.784,-176.820,11.385,149.493
C03267=1132.326,398.346,-88.820,-176.820,11.388,149.494
C03268=1132.322,398.594,-88.859,-176.820,11.391,149.494
C03269=1132.318,398.840,-88.897,-176.819,11.393,149.495
C03270=1132.315,399.088,-88.934,-176.820,11.396,149.496
C03271=1132.311,399.334,-88.972,-176.820,11.399,149.497
C03272=1132.307,399.582,-89.011,-176.820,11.401,149.497
C03273=1132.304,399.828,-89.048,-176.820,11.404,149.498
C03274=1132.300,400.076,-89.086,-176.820,11.407,149.499
C03275=1132.296,400.323,-89.124,-176.819,11.410,149.499
C03276=1132.293,400.570,-89.162,-176.820,11.413,149.500
C03277=1132.289,400.817,-89.200,-176.820,11.416,149.501
C03278=1132.285,401.064,-89.238,-176.820,11.418,149.502
C03279=1132.282,401.311,-89.276,-176.820,11.421,149.503
C03280=1132.278,401.558,-89.314,-176.820,11.424,149.503
C03281=1132.275,401.805,-89.352,-176.820,11.428,149.504
C03282=1132.270,402.052,-89.390,-176.820,11.430,149.505
C03283=1132.267,402.265,-89.423,-176.820,11.433,149.506
C03284=1132.264,402.477,-89.455,-176.821,11.435,149.506
C03285=1132.261,402.689,-89.487,-176.821,11.438,149.507
C03286=1132.258,402.903,-89.520,-176.821,11.440,149.508
C03287=1132.255,403.115,-89.553,-176.821,11.443,149.509
C03288=1132.251,403.327,-89.586,-176.822,11.446,149.509
C03289=1132.248,403.540,-89.619,-176.822,11.449,149.510
C03290=1132.245,403.753,-89.651,-176.822,11.451,149.511
C03291=1132.242,404.000,-89.689,-176.823,11.455,149.512
C03292=1132.237,404.247,-89.727,-176.823,11.458,149.513
C03293=1132.234,404.494,-89.765,-176.823,11.462,149.514
C03294=1132.230,404.741,-89.803,-176.823,11.464,149.515
C03295=1132.226,404.988,-89.841,-176.824,11.468,149.516
C03296=1132.223,405.235,-89.879,-176.825,11.471,149.517
C03297=1132.219,405.482,-89.917,-176.825,11.475,149.518
C03298=1132.215,405.730,-89.955,-176.825,11.478,149.519
C03299=1132.212,405.976,-89.993,-176.826,11.481,149.520
C03300=1132.208,406.224,-90.031,-176.826,11.485,149.521
C03301=1132.205,406.471,-90.069,-176.827,11.488,149.522
C03302=1132.201,406.718,-90.107,-176.827,11.491,149.523
C03303=1132.197,406.965,-90.146,-176.829,11.495,149.524
C03304=1132.193,407.212,-90.183,-176.829,11.499,149.525
C03305=1132.190,407.459,-90.221,-176.829,11.502,149.526
C03306=1132.186,407.707,-90.260,-176.830,11.506,149.527
C03307=1132.182,407.953,-90.298,-176.831,11.510,149.528
C03308=1132.178,408.200,-90.336,-176.832,11.513,149.529
C03309=1132.175,408.447,-90.374,-176.832,11.517,149.530
C03310=1132.172,408.694,-90.412,-176.833,11.521,149.532
C03311=1132.168,408.942,-90.450,-176.834,11.524,149.533
C03312=1132.164,409.188,-90.488,-176.834,11.528,149.534
C03313=1132.160,409.436,-90.527,-176.835,11.532,149.535
C03314=1132.156,409.682,-90.564,-176.836,11.535,149.536
C03315=1132.153,409.930,-90.602,-176.837,11.540,149.538
C03316=1132.149,410.176,-90.641,-176.838,11.543,149.539
C03317=1132.145,410.423,-90.679,-176.839,11.548,149.540
C03318=1132.142,410.671,-90.717,-176.840,11.552,149.541
C03319=1132.138,410.917,-90.755,-176.840,11.556,149.543
C03320=1132.135,411.164,-90.793,-176.842,11.560,149.544
C03321=1132.131,411.412,-90.831,-176.843,11.563,149.545
C03322=1132.127,411.659,-90.869,-176.843,11.568,149.547
C03323=1132.123,411.906,-90.908,-176.845,11.571,149.548
C03324=1132.119,412.152,-90.946,-176.845,11.576,149.549
C03325=1132.116,412.400,-90.984,-176.847,11.580,149.551
C03326=1132.112,412.647,-91.022,-176.848,11.585,149.552
C03327=1132.109,412.894,-91.060,-176.849,11.588,149.553
C03328=1132.105,413.141,-91.098,-176.850,11.593,149.555
C03329=1132.101,413.388,-91.136,-176.851,11.597,149.556
C03330=1132.097,413.635,-91.175,-176.852,11.602,149.558
C03331=1132.094,413.882,-91.213,-176.853,11.606,149.559
C03332=1132.090,414.129,-91.251,-176.855,11.610,149.560
C03333=1132.086,414.376,-91.289,-176.856,11.615,149.562
C03334=1132.085,414.623,-91.328,-176.857,11.619,149.563
C03335=1132.082,414.870,-91.366,-176.859,11.624,149.565
C03336=1132.081,415.117,-91.404,-176.860,11.628,149.566
C03337=1132.080,415.364,-91.441,-176.861,11.633,149.568
C03338=1132.079,415.612,-91.479,-176.863,11.637,149.570
C03339=1132.080,415.824,-91.511,-176.864,11.642,149.571
C03340=1132.081,416.037,-91.544,-176.865,11.645,149.572
C03341=1132.082,416.248,-91.576,-176.866,11.649,149.574
C03342=1132.083,416.461,-91.608,-176.868,11.653,149.575
C03343=1132.086,416.674,-91.640,-176.869,11.657,149.576
C03344=1132.088,416.886,-91.673,-176.870,11.662,149.578
C03345=1132.091,417.099,-91.704,-176.872,11.666,149.579
C03346=1132.095,417.311,-91.736,-176.874,11.670,149.581
C03347=1131.676,417.311,-91.799,-176.866,11.674,149.580
C03348=1131.672,417.099,-91.767,-176.865,11.670,149.579
C03349=1131.669,416.886,-91.735,-176.863,11.666,149.577
C03350=1131.666,416.673,-91.703,-176.862,11.662,149.576
C03351=1131.665,416.461,-91.671,-176.861,11.658,149.574
C03352=1131.663,416.248,-91.639,-176.859,11.654,149.573
C03353=1131.661,416.036,-91.606,-176.858,11.650,149.572
C03354=1131.661,415.824,-91.574,-176.857,11.645,149.570
C03355=1131.661,415.612,-91.542,-176.856,11.641,149.569
C03356=1131.661,415.365,-91.503,-176.854,11.637,149.567
C03357=1131.662,415.117,-91.466,-176.853,11.633,149.566
C03358=1131.663,414.870,-91.428,-176.852,11.628,149.564
C03359=1131.665,414.623,-91.389,-176.850,11.624,149.563
C03360=1131.667,414.376,-91.352,-176.849,11.619,149.561
C03361=1131.671,414.129,-91.314,-176.848,11.614,149.560
C03362=1131.674,413.882,-91.275,-176.847,11.610,149.558
C03363=1131.678,413.635,-91.237,-176.846,11.606,149.557
C03364=1131.682,413.388,-91.199,-176.844,11.601,149.555
C03365=1131.685,413.140,-91.161,-176.843,11.597,149.554
C03366=1131.690,412.894,-91.123,-176.842,11.592,149.553
C03367=1131.693,412.647,-91.084,-176.841,11.588,149.551
C03368=1131.696,412.400,-91.046,-176.841,11.584,149.550
C03369=1131.700,412.153,-91.008,-176.839,11.580,149.549
C03370=1131.703,411.905,-90.970,-176.838,11.575,149.547
C03371=1131.708,411.659,-90.932,-176.837,11.572,149.546
C03372=1131.711,411.411,-90.894,-176.836,11.567,149.545
C03373=1131.715,411.164,-90.855,-176.835,11.564,149.543
C03374=1131.719,410.918,-90.817,-176.835,11.559,149.542
C03375=1131.722,410.670,-90.778,-176.833,11.555,149.541
C03376=1131.726,410.423,-90.741,-176.833,11.551,149.540
C03377=1131.729,410.176,-90.703,-176.832,11.547,149.538
C03378=1131.733,409.929,-90.664,-176.831,11.543,149.537
C03379=1131.737,409.683,-90.626,-176.830,11.540,149.536
C03380=1131.741,409.435,-90.588,-176.830,11.535,149.535
C03381=1131.744,409.188,-90.550,-176.829,11.532,149.533
C03382=1131.748,408.941,-90.512,-176.828,11.527,149.532
C03383=1131.752,408.694,-90.474,-176.827,11.524,149.531
C03384=1131.755,408.447,-90.436,-176.827,11.520,149.530
C03385=1131.759,408.200,-90.397,-176.826,11.516,149.529
C03386=1131.763,407.952,-90.360,-176.825,11.513,149.528
C03387=1131.766,407.706,-90.321,-176.825,11.509,149.526
C03388=1131.770,407.459,-90.283,-176.824,11.506,149.525
C03389=1131.774,407.212,-90.245,-176.824,11.502,149.524
C03390=1131.778,406.965,-90.207,-176.823,11.498,149.523
C03391=1131.781,406.717,-90.169,-176.822,11.495,149.522
C03392=1131.785,406.471,-90.131,-176.822,11.491,149.521
C03393=1131.789,406.223,-90.093,-176.821,11.488,149.520
C03394=1131.792,405.977,-90.055,-176.821,11.484,149.519
C03395=1131.796,405.729,-90.016,-176.821,11.480,149.518
C03396=1131.799,405.482,-89.978,-176.820,11.478,149.517
C03397=1131.803,405.235,-89.941,-176.820,11.474,149.516
C03398=1131.807,404.988,-89.902,-176.819,11.470,149.515
C03399=1131.811,404.741,-89.865,-176.819,11.467,149.514
C03400=1131.814,404.495,-89.826,-176.818,11.464,149.513
C03401=1131.818,404.247,-89.788,-176.818,11.460,149.512
C03402=1131.822,404.000,-89.750,-176.818,11.457,149.511
C03403=1131.825,403.753,-89.712,-176.818,11.454,149.511
C03404=1131.828,403.541,-89.680,-176.817,11.452,149.510
C03405=1131.832,403.328,-89.647,-176.817,11.449,149.509
C03406=1131.835,403.115,-89.614,-176.817,11.446,149.508
C03407=1131.838,402.903,-89.581,-176.817,11.443,149.507
C03408=1131.841,402.690,-89.548,-176.817,11.441,149.507
C03409=1131.844,402.478,-89.516,-176.817,11.438,149.506
C03410=1131.848,402.265,-89.483,-176.817,11.435,149.505
C03411=1131.851,402.052,-89.450,-176.816,11.432,149.505
C03412=1131.855,401.806,-89.413,-176.816,11.429,149.504
C03413=1131.858,401.558,-89.375,-176.816,11.427,149.503
C03414=1131.862,401.312,-89.337,-176.816,11.423,149.502
C03415=1131.865,401.064,-89.299,-176.816,11.420,149.501
C03416=1131.869,400.818,-89.261,-176.816,11.418,149.501
C03417=1131.873,400.570,-89.223,-176.816,11.415,149.500
C03418=1131.877,400.324,-89.185,-176.816,11.412,149.499
C03419=1131.880,400.076,-89.147,-176.816,11.409,149.498
C03420=1131.884,399.829,-89.109,-176.816,11.406,149.498
C03421=1131.888,399.582,-89.071,-176.816,11.403,149.497
C03422=1131.891,399.335,-89.033,-176.816,11.401,149.496
C03423=1131.895,399.088,-88.995,-176.816,11.398,149.496
C03424=1131.899,398.840,-88.958,-176.816,11.396,149.495
C03425=1131.903,398.593,-88.920,-176.817,11.392,149.494
C03426=1131.906,398.346,-88.882,-176.817,11.390,149.494
C03427=1131.911,398.099,-88.844,-176.817,11.387,149.493
C03428=1131.914,397.852,-88.806,-176.817,11.385,149.492
C03429=1131.918,397.606,-88.768,-176.817,11.382,149.492
C03430=1131.921,397.358,-88.730,-176.817,11.379,149.491
C03431=1131.925,397.111,-88.692,-176.818,11.376,149.490
C03432=1131.928,396.864,-88.654,-176.818,11.374,149.490
C03433=1131.932,396.618,-88.617,-176.818,11.371,149.489
C03434=1131.936,396.369,-88.579,-176.819,11.369,149.489
C03435=1131.940,396.123,-88.541,-176.819,11.367,149.488
C03436=1131.943,395.875,-88.503,-176.819,11.364,149.487
C03437=1131.947,395.629,-88.466,-176.820,11.362,149.487
C03438=1131.951,395.381,-88.427,-176.820,11.360,149.487
C03439=1131.954,395.134,-88.389,-176.820,11.357,149.486
C03440=1131.958,394.887,-88.352,-176.821,11.354,149.485
C03441=1131.962,394.640,-88.315,-176.822,11.352,149.485
C03442=1131.966,394.393,-88.276,-176.822,11.349,149.484
C03443=1131.970,394.146,-88.239,-176.823,11.347,149.484
C03444=1131.973,393.899,-88.201,-176.823,11.345,149.484
C03445=1131.977,393.652,-88.163,-176.823,11.343,149.483
C03446=1131.981,393.405,-88.125,-176.824,11.341,149.483
C03447=1131.985,393.158,-88.088,-176.824,11.338,149.482
C03448=1131.988,392.910,-88.050,-176.825,11.336,149.482
C03449=1131.992,392.664,-88.012,-176.825,11.334,149.481
C03450=1131.995,392.416,-87.975,-176.826,11.332,149.481
C03451=1132.000,392.169,-87.937,-176.827,11.330,149.480
C03452=1132.003,391.922,-87.899,-176.827,11.328,149.480
C03453=1132.007,391.675,-87.862,-176.828,11.326,149.480
C03454=1132.010,391.428,-87.824,-176.829,11.323,149.479
C03455=1132.014,391.181,-87.786,-176.830,11.321,149.479
C03456=1132.018,390.933,-87.748,-176.830,11.318,149.479
C03457=1132.022,390.686,-87.711,-176.831,11.317,149.478
C03458=1132.025,390.439,-87.673,-176.832,11.315,149.478
C03459=1132.029,390.193,-87.635,-176.833,11.313,149.478
C03460=1132.032,389.979,-87.603,-176.833,11.311,149.477
C03461=1132.036,389.767,-87.570,-176.834,11.309,149.477
C03462=1132.038,389.555,-87.538,-176.834,11.308,149.477
C03463=1132.041,389.342,-87.505,-176.836,11.306,149.477
C03464=1132.045,389.129,-87.473,-176.836,11.305,149.476
C03465=1132.048,388.916,-87.441,-176.837,11.303,149.476
C03466=1132.051,388.704,-87.409,-176.838,11.301,149.476
C03467=1132.054,388.491,-87.376,-176.839,11.299,149.476
C03468=1132.058,388.244,-87.339,-176.839,11.297,149.475
C03469=1132.061,387.997,-87.301,-176.840,11.295,149.475
C03470=1132.066,387.750,-87.263,-176.841,11.294,149.475
C03471=1132.070,387.503,-87.226,-176.842,11.292,149.475
C03472=1132.073,387.255,-87.188,-176.843,11.290,149.474
C03473=1132.077,387.009,-87.151,-176.844,11.288,149.474
C03474=1132.080,386.761,-87.113,-176.845,11.286,149.474
C03475=1132.084,386.514,-87.076,-176.846,11.285,149.474
C03476=1132.087,386.267,-87.038,-176.847,11.283,149.474
C03477=1132.091,386.020,-87.001,-176.848,11.281,149.473
C03478=1132.095,385.772,-86.962,-176.850,11.280,149.473
C03479=1132.100,385.525,-86.926,-176.851,11.278,149.473
C03480=1132.103,385.278,-86.888,-176.852,11.276,149.473
C03481=1132.106,385.031,-86.850,-176.853,11.274,149.473
C03482=1132.111,384.784,-86.813,-176.854,11.273,149.473
C03483=1132.114,384.537,-86.775,-176.855,11.271,149.472
C03484=1132.118,384.290,-86.738,-176.856,11.269,149.472
C03485=1132.122,384.043,-86.701,-176.857,11.268,149.472
C03486=1132.125,383.796,-86.663,-176.859,11.266,149.472
C03487=1132.129,383.549,-86.626,-176.860,11.265,149.472
C03488=1132.132,383.301,-86.588,-176.861,11.263,149.472
C03489=1132.136,383.054,-86.551,-176.864,11.260,149.472
C03490=1132.140,382.806,-86.513,-176.867,11.259,149.472
C03491=1132.144,382.559,-86.476,-176.870,11.256,149.472
C03492=1132.148,382.313,-86.438,-176.872,11.254,149.472
C03493=1132.152,382.065,-86.401,-176.874,11.252,149.472
C03494=1132.155,381.818,-86.364,-176.877,11.249,149.472
C03495=1132.159,381.571,-86.327,-176.879,11.247,149.472
C03496=1132.163,381.324,-86.289,-176.882,11.244,149.473
C03497=1132.167,381.077,-86.252,-176.885,11.242,149.473
C03498=1132.171,380.829,-86.215,-176.888,11.240,149.473
C03499=1132.174,380.582,-86.177,-176.890,11.238,149.473
C03500=1132.178,380.335,-86.140,-176.893,11.235,149.473
C03501=1132.181,380.088,-86.102,-176.896,11.233,149.473
C03502=1132.185,379.841,-86.065,-176.899,11.230,149.473
C03503=1132.189,379.593,-86.029,-176.901,11.228,149.473
C03504=1132.193,379.346,-85.991,-176.904,11.226,149.473
C03505=1132.197,379.099,-85.954,-176.906,11.224,149.473
C03506=1132.200,378.852,-85.917,-176.909,11.221,149.473
C03507=1132.204,378.605,-85.880,-176.912,11.219,149.474
C03508=1132.207,378.358,-85.843,-176.915,11.216,149.474
C03509=1132.211,378.110,-85.806,-176.918,11.215,149.474
C03510=1132.215,377.864,-85.768,-176.920,11.212,149.474
C03511=1132.219,377.616,-85.731,-176.923,11.210,149.474
C03512=1132.223,377.369,-85.694,-176.926,11.207,149.474
C03513=1132.227,377.121,-85.657,-176.929,11.206,149.474
C03514=1132.230,376.874,-85.619,-176.932,11.203,149.474
C03515=1132.234,376.627,-85.583,-176.934,11.201,149.475
C03516=1132.237,376.414,-85.551,-176.937,11.199,149.475
C03517=1132.241,376.201,-85.519,-176.939,11.197,149.475
C03518=1132.244,375.989,-85.487,-176.942,11.195,149.475
C03519=1132.248,375.776,-85.456,-176.944,11.193,149.475
C03520=1132.250,375.563,-85.424,-176.947,11.191,149.475
C03521=1132.253,375.351,-85.391,-176.949,11.189,149.475
C03522=1132.257,375.138,-85.360,-176.952,11.187,149.475
C03523=1132.260,374.925,-85.328,-176.954,11.185,149.476
C03524=1132.264,374.678,-85.292,-176.958,11.183,149.476
C03525=1132.268,374.431,-85.255,-176.960,11.181,149.476
C03526=1132.271,374.183,-85.218,-176.963,11.178,149.476
C03527=1132.275,373.936,-85.181,-176.966,11.176,149.476
C03528=1132.279,373.689,-85.144,-176.969,11.174,149.476
C03529=1132.283,373.442,-85.108,-176.972,11.171,149.477
C03530=1132.286,373.194,-85.071,-176.975,11.169,149.477
C03531=1132.290,372.947,-85.033,-176.978,11.167,149.477
C03532=1132.294,372.700,-84.996,-176.981,11.164,149.477
C03533=1132.298,372.453,-84.960,-176.984,11.163,149.477
C03534=1132.302,372.206,-84.924,-176.987,11.160,149.478
C03535=1132.305,371.958,-84.887,-176.990,11.158,149.478
C03536=1132.309,371.711,-84.850,-176.993,11.156,149.478
C03537=1132.313,371.464,-84.813,-176.996,11.153,149.478
C03538=1132.317,371.216,-84.777,-176.999,11.151,149.478
C03539=1132.321,370.969,-84.740,-177.002,11.149,149.478
C03540=1132.324,370.722,-84.703,-177.005,11.146,149.479
C03541=1132.328,370.474,-84.666,-177.008,11.144,149.479
C03542=1132.332,370.227,-84.629,-177.011,11.142,149.479
C03543=1132.335,369.980,-84.593,-177.014,11.140,149.479
C03544=1132.339,369.733,-84.556,-177.018,11.137,149.480
C03545=1132.344,369.485,-84.520,-177.021,11.135,149.480
C03546=1132.347,369.238,-84.484,-177.024,11.133,149.480
C03547=1132.351,368.991,-84.447,-177.027,11.131,149.480
C03548=1132.354,368.744,-84.410,-177.030,11.128,149.480
C03549=1132.358,368.496,-84.374,-177.033,11.126,149.481
C03550=1132.363,368.249,-84.337,-177.036,11.124,149.481
C03551=1132.366,368.002,-84.301,-177.039,11.122,149.481
C03552=1132.370,367.755,-84.264,-177.043,11.119,149.481
C03553=1132.374,367.507,-84.229,-177.046,11.117,149.482
C03554=1132.378,367.260,-84.192,-177.049,11.115,149.482
C03555=1132.381,367.013,-84.156,-177.052,11.112,149.482
C03556=1132.386,366.765,-84.119,-177.055,11.110,149.482
C03557=1132.390,366.518,-84.083,-177.059,11.107,149.482
C03558=1132.393,366.271,-84.046,-177.062,11.105,149.483
C03559=1132.397,366.023,-84.010,-177.065,11.103,149.483
C03560=1132.400,365.776,-83.973,-177.068,11.101,149.483
C03561=1132.404,365.529,-83.937,-177.072,11.099,149.483
C03562=1132.408,365.281,-83.901,-177.075,11.096,149.484
C03563=1132.412,365.034,-83.864,-177.078,11.094,149.484
C03564=1132.416,364.786,-83.829,-177.082,11.091,149.484
C03565=1132.420,364.539,-83.792,-177.085,11.089,149.484
C03566=1132.423,364.292,-83.756,-177.088,11.086,149.485
C03567=1132.427,364.045,-83.720,-177.091,11.084,149.485
C03568=1132.431,363.797,-83.684,-177.095,11.082,149.485
C03569=1132.435,363.550,-83.648,-177.098,11.080,149.485
C03570=1132.439,363.302,-83.611,-177.101,11.078,149.486
C03571=1132.442,363.055,-83.575,-177.104,11.075,149.486
C03572=1132.446,362.842,-83.545,-177.108,11.073,149.486
C03573=1132.449,362.629,-83.513,-177.110,11.071,149.486
C03574=1132.452,362.417,-83.482,-177.114,11.068,149.487
C03575=1132.455,362.204,-83.452,-177.116,11.067,149.487
C03576=1132.459,361.991,-83.420,-177.119,11.065,149.487
C03577=1132.462,361.777,-83.389,-177.122,11.063,149.487
C03578=1132.465,361.565,-83.358,-177.125,11.061,149.487
C03579=1132.468,361.352,-83.327,-177.128,11.058,149.488
C03580=1132.472,361.104,-83.291,-177.132,11.056,149.488
C03581=1132.476,360.857,-83.255,-177.135,11.054,149.488
C03582=1132.480,360.611,-83.219,-177.138,11.051,149.488
C03583=1132.484,360.363,-83.183,-177.142,11.049,149.489
C03584=1132.488,360.116,-83.148,-177.145,11.046,149.489
C03585=1132.492,359.868,-83.112,-177.149,11.044,149.489
C03586=1132.495,359.621,-83.075,-177.152,11.042,149.489
C03587=1132.499,359.373,-83.040,-177.155,11.039,149.490
C03588=1132.503,359.125,-83.004,-177.159,11.037,149.490
C03589=1132.507,358.878,-82.968,-177.162,11.034,149.490
C03590=1132.511,358.630,-82.933,-177.166,11.032,149.491
C03591=1132.514,358.384,-82.896,-177.169,11.030,149.491
C03592=1132.518,358.136,-82.861,-177.173,11.027,149.491
C03593=1132.522,357.888,-82.825,-177.176,11.024,149.491
C03594=1132.526,357.642,-82.790,-177.180,11.022,149.492
C03595=1132.530,357.394,-82.754,-177.183,11.020,149.492
C03596=1132.534,357.147,-82.718,-177.187,11.017,149.492
C03597=1132.537,356.899,-82.683,-177.190,11.015,149.492
C03598=1132.542,356.651,-82.647,-177.194,11.011,149.493
C03599=1132.546,356.404,-82.611,-177.198,11.009,149.493
C03600=1132.549,356.156,-82.576,-177.201,11.007,149.493
C03601=1132.553,355.909,-82.540,-177.204,11.004,149.493
C03602=1132.557,355.662,-82.505,-177.208,11.002,149.494
C03603=1132.561,355.414,-82.469,-177.212,10.999,149.494
C03604=1132.564,355.167,-82.434,-177.215,10.996,149.494
C03605=1132.569,354.919,-82.398,-177.219,10.994,149.495
C03606=1132.573,354.672,-82.362,-177.222,10.992,149.495
C03607=1132.577,354.425,-82.327,-177.226,10.989,149.495
C03608=1132.580,354.177,-82.291,-177.230,10.986,149.495
C03609=1132.584,353.930,-82.256,-177.233,10.984,149.496
C03610=1132.588,353.682,-82.220,-177.237,10.982,149.496
C03611=1132.591,353.435,-82.185,-177.241,10.978,149.496
C03612=1132.596,353.188,-82.150,-177.244,10.976,149.497
C03613=1132.600,352.940,-82.115,-177.248,10.974,149.497
C03614=1132.603,352.692,-82.079,-177.251,10.970,149.497
C03615=1132.607,352.445,-82.044,-177.255,10.968,149.497
C03616=1132.611,352.198,-82.008,-177.259,10.965,149.498
C03617=1132.615,351.951,-81.973,-177.262,10.963,149.498
C03618=1132.619,351.702,-81.938,-177.266,10.961,149.498
C03619=1132.623,351.455,-81.903,-177.270,10.957,149.498
C03620=1132.627,351.208,-81.867,-177.273,10.955,149.499
C03621=1132.631,350.960,-81.833,-177.277,10.952,149.499
C03622=1132.634,350.713,-81.797,-177.281,10.949,149.499
C03623=1132.639,350.466,-81.762,-177.284,10.947,149.499
C03624=1132.643,350.218,-81.727,-177.288,10.944,149.500
C03625=1132.646,349.970,-81.691,-177.292,10.942,149.500
C03626=1132.651,349.723,-81.656,-177.296,10.938,149.500
C03627=1132.655,349.475,-81.621,-177.299,10.936,149.500
C03628=1132.657,349.262,-81.591,-177.303,10.933,149.501
C03629=1132.661,349.049,-81.561,-177.305,10.931,149.501
C03630=1132.664,348.836,-81.531,-177.308,10.929,149.501
C03631=1132.667,348.623,-81.501,-177.311,10.927,149.501
C03632=1132.671,348.409,-81.471,-177.313,10.925,149.501
C03633=1132.675,348.197,-81.441,-177.316,10.923,149.502
C03634=1132.678,347.984,-81.410,-177.319,10.921,149.502
C03635=1132.681,347.771,-81.380,-177.322,10.918,149.502
C03636=1132.685,347.523,-81.346,-177.325,10.916,149.502
C03637=1132.689,347.276,-81.310,-177.329,10.913,149.502
C03638=1132.693,347.028,-81.275,-177.332,10.911,149.503
C03639=1132.697,346.781,-81.240,-177.335,10.909,149.503
C03640=1132.700,346.533,-81.206,-177.339,10.906,149.503
C03641=1132.705,346.286,-81.171,-177.342,10.903,149.503
C03642=1132.709,346.038,-81.136,-177.345,10.901,149.503
C03643=1132.713,345.790,-81.101,-177.348,10.898,149.503
C03644=1132.716,345.544,-81.066,-177.351,10.896,149.504
C03645=1132.720,345.295,-81.032,-177.354,10.894,149.504
C03646=1132.725,345.048,-80.997,-177.357,10.892,149.504
